KUKA KRL program: f1_Kuka_APT207T03S07.SRC

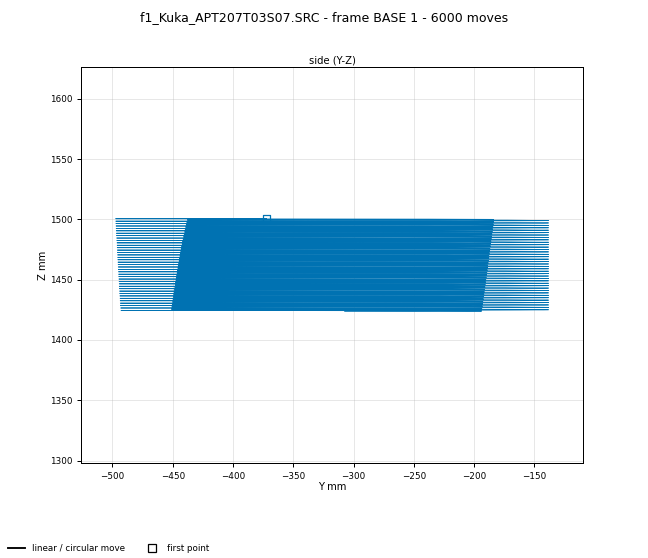
[picture p0: tool path of f1_Kuka_APT207T03S07.SRC in frame BASE 1, 6000 of 6001 moves have a stored position in this frame; points joined in program order, loops and branches not executed]
&ACCESS RVP
&REL 2
&PARAM TEMPLATE = C:\KRC\Roboter\Template\vorgabe
&PARAM EDITMASK = *
DEF f1_Kuka_APT207T03S07()


;FOLD INI;%{PE}%V3.2.0,%MKUKATPBASIS,%CINIT,%VCOMMON,%P
  ;FOLD BAS INI;%{E}%V3.2.0,%MKUKATPBASIS,%CINIT,%VINIT,%P
    GLOBAL INTERRUPT DECL 3 WHEN $STOPMESS==TRUE DO IR_STOPM ( )
    INTERRUPT ON 3
    BAS (#INITMOV,0 )
  ;ENDFOLD (BAS INI)
  ;FOLD USER INI;%{E}%V3.2.0,%MKUKATPUSER,%CINIT,%VINIT,%P
    ;Make your modifications here
  ;ENDFOLD (USER INI)
;ENDFOLD (INI)


;*** Make Null PTP Move
  PTP $pos_act

;*** Auto Load The Correct TOOL Data
  $tool=tool_data[3]

;*** Auto Load The Correct BASE Data
  $base=base_data[1]

  $ADVANCE = 5

;*** Restate Last Velocity
MMPM(30000.0)
SetRPM(6000)
LIN {X 0.159,Y -372.201,Z 1500.629,A 0.000,B 0.000,C 90.000,E1 113.206} C_DIS
LIN {X -0.112,Y -386.220,Z 1500.616,A 0.000,B 0.000,C 90.000,E1 110.918} C_DIS
LIN {X 0.185,Y -401.630,Z 1500.604,A 0.000,B 0.000,C 90.000,E1 108.598} C_DIS
LIN {X 0.113,Y -418.538,Z 1500.591,A 0.000,B 0.000,C 90.000,E1 106.386} C_DIS
LIN {X -0.068,Y -437.063,Z 1500.579,A 0.000,B 0.000,C 90.000,E1 104.245} C_DIS
LIN {X -0.031,Y -456.906,Z 1500.568,A 0.000,B 0.000,C 90.000,E1 102.175} C_DIS
LIN {X 0.162,Y -477.322,Z 1500.557,A 0.000,B 0.000,C 90.000,E1 100.254} C_DIS
LIN {X 0.127,Y -490.260,Z 1500.551,A 0.000,B 0.000,C 90.000,E1 99.151} C_DIS
LIN {X -0.192,Y -492.261,Z 1500.550,A 0.000,B 0.000,C 90.000,E1 98.973} C_DIS
LIN {X 0.126,Y -493.981,Z 1500.548,A 0.000,B 0.000,C 90.000,E1 98.690} C_DIS
LIN {X 0.030,Y -495.267,Z 1500.547,A 0.000,B 0.000,C 90.000,E1 98.454} C_DIS
LIN {X -0.213,Y -496.844,Z 1500.544,A 0.000,B 0.000,C 90.000,E1 97.992} C_DIS
LIN {X 0.043,Y -497.342,Z 1500.542,A 0.000,B 0.000,C 90.000,E1 97.473} C_DIS
LIN {X -0.122,Y -496.847,Z 1500.539,A 0.000,B 0.000,C 90.000,E1 97.004} C_DIS
LIN {X 0.144,Y -495.281,Z 1500.536,A 0.000,B 0.000,C 90.000,E1 96.486} C_DIS
LIN {X 0.002,Y -494.010,Z 1500.535,A 0.000,B 0.000,C 90.000,E1 96.258} C_DIS
LIN {X 0.215,Y -484.168,Z 1500.527,A 0.000,B 0.000,C 90.000,E1 94.759} C_DIS
LIN {X 0.034,Y -473.583,Z 1500.517,A 0.000,B 0.000,C 90.000,E1 93.037} C_DIS
LIN {X 0.219,Y -467.179,Z 1500.511,A 0.000,B 0.000,C 90.000,E1 92.007} C_DIS
LIN {X -0.087,Y -457.018,Z 1500.503,A 0.000,B 0.000,C 90.000,E1 90.516} C_DIS
LIN {X -0.114,Y -446.557,Z 1500.494,A 0.000,B 0.000,C 90.000,E1 88.969} C_DIS
LIN {X 0.127,Y -435.874,Z 1500.485,A 0.000,B 0.000,C 90.000,E1 87.364} C_DIS
LIN {X 0.018,Y -421.489,Z 1500.474,A 0.000,B 0.000,C 90.000,E1 85.241} C_DIS
LIN {X -0.123,Y -410.754,Z 1500.464,A 0.000,B 0.000,C 90.000,E1 83.628} C_DIS
LIN {X 0.119,Y -396.318,Z 1500.452,A 0.000,B 0.000,C 90.000,E1 81.376} C_DIS
LIN {X -0.155,Y -377.030,Z 1500.435,A 0.000,B 0.000,C 90.000,E1 78.285} C_DIS
LIN {X -0.065,Y -363.896,Z 1500.422,A 0.000,B 0.000,C 90.000,E1 75.936} C_DIS
LIN {X -0.051,Y -352.647,Z 1500.410,A 0.000,B 0.000,C 90.000,E1 73.850} C_DIS
LIN {X 0.045,Y -341.368,Z 1500.398,A 0.000,B 0.000,C 90.000,E1 71.710} C_DIS
LIN {X -0.125,Y -328.685,Z 1500.385,A 0.000,B 0.000,C 90.000,E1 69.263} C_DIS
LIN {X 0.116,Y -313.654,Z 1500.367,A 0.000,B 0.000,C 90.000,E1 66.049} C_DIS
LIN {X 0.098,Y -300.896,Z 1500.351,A 0.000,B 0.000,C 90.000,E1 63.127} C_DIS
LIN {X 0.137,Y -288.807,Z 1500.334,A 0.000,B 0.000,C 90.000,E1 60.127} C_DIS
LIN {X -0.069,Y -278.507,Z 1500.319,A 0.000,B 0.000,C 90.000,E1 57.454} C_DIS
LIN {X -0.074,Y -268.552,Z 1500.304,A 0.000,B 0.000,C 90.000,E1 54.689} C_DIS
LIN {X 0.138,Y -258.980,Z 1500.288,A 0.000,B 0.000,C 90.000,E1 51.823} C_DIS
LIN {X 0.047,Y -248.766,Z 1500.270,A 0.000,B 0.000,C 90.000,E1 48.609} C_DIS
LIN {X -0.011,Y -238.232,Z 1500.250,A 0.000,B 0.000,C 90.000,E1 44.960} C_DIS
LIN {X -0.114,Y -230.557,Z 1500.233,A 0.000,B 0.000,C 90.000,E1 42.000} C_DIS
LIN {X -0.005,Y -222.002,Z 1500.212,A 0.000,B 0.000,C 90.000,E1 38.177} C_DIS
LIN {X -0.052,Y -214.472,Z 1500.191,A 0.000,B 0.000,C 90.000,E1 34.326} C_DIS
LIN {X 0.012,Y -207.800,Z 1500.169,A 0.000,B 0.000,C 90.000,E1 30.384} C_DIS
LIN {X -0.013,Y -202.023,Z 1500.147,A 0.000,B 0.000,C 90.000,E1 26.411} C_DIS
LIN {X -0.024,Y -197.120,Z 1500.124,A 0.000,B 0.000,C 90.000,E1 22.386} C_DIS
LIN {X 0.001,Y -192.945,Z 1500.102,A 0.000,B 0.000,C 90.000,E1 18.308} C_DIS
LIN {X 0.065,Y -188.915,Z 1500.074,A 0.000,B 0.000,C 90.000,E1 13.355} C_DIS
LIN {X -0.062,Y -185.704,Z 1500.042,A 0.000,B 0.000,C 90.000,E1 7.587} C_DIS
LIN {X 0.089,Y -183.811,Z 1500.005,A 0.000,B 0.000,C 90.000,E1 0.859} C_DIS
LIN {X -0.056,Y -183.944,Z 1499.965,A 0.000,B 0.000,C 90.000,E1 353.685} C_DIS
LIN {X -0.092,Y -186.302,Z 1499.923,A 0.000,B 0.000,C 90.000,E1 346.172} C_DIS
LIN {X 0.027,Y -189.401,Z 1499.895,A 0.000,B 0.000,C 90.000,E1 341.148} C_DIS
LIN {X -0.076,Y -193.715,Z 1499.868,A 0.000,B 0.000,C 90.000,E1 336.230} C_DIS
LIN {X 0.063,Y -198.267,Z 1499.845,A 0.000,B 0.000,C 90.000,E1 332.103} C_DIS
LIN {X 0.013,Y -203.831,Z 1499.823,A 0.000,B 0.000,C 90.000,E1 328.074} C_DIS
LIN {X -0.061,Y -209.063,Z 1499.805,A 0.000,B 0.000,C 90.000,E1 324.895} C_DIS
LIN {X 0.071,Y -215.145,Z 1499.787,A 0.000,B 0.000,C 90.000,E1 321.698} C_DIS
LIN {X -0.048,Y -222.035,Z 1499.770,A 0.000,B 0.000,C 90.000,E1 318.609} C_DIS
LIN {X -0.009,Y -229.890,Z 1499.753,A 0.000,B 0.000,C 90.000,E1 315.526} C_DIS
LIN {X -0.087,Y -238.715,Z 1499.736,A 0.000,B 0.000,C 90.000,E1 312.528} C_DIS
LIN {X -0.073,Y -249.962,Z 1499.718,A 0.000,B 0.000,C 90.000,E1 309.197} C_DIS
LIN {X 0.003,Y -257.116,Z 1499.708,A 0.000,B 0.000,C 90.000,E1 307.363} C_DIS
LIN {X -0.111,Y -265.197,Z 1499.698,A 0.000,B 0.000,C 90.000,E1 305.598} C_DIS
LIN {X 0.122,Y -274.179,Z 1499.688,A 0.000,B 0.000,C 90.000,E1 303.785} C_DIS
LIN {X -0.024,Y -284.237,Z 1499.678,A 0.000,B 0.000,C 90.000,E1 302.084} C_DIS
LIN {X -0.031,Y -297.487,Z 1499.667,A 0.000,B 0.000,C 90.000,E1 300.050} C_DIS
LIN {X 0.119,Y -307.294,Z 1499.660,A 0.000,B 0.000,C 90.000,E1 298.693} C_DIS
LIN {X 0.060,Y -328.798,Z 1499.646,A 0.000,B 0.000,C 90.000,E1 296.181} C_DIS
LIN {X -0.035,Y -347.607,Z 1499.634,A 0.000,B 0.000,C 90.000,E1 294.207} C_DIS
LIN {X -0.091,Y -363.609,Z 1499.625,A 0.000,B 0.000,C 90.000,E1 292.589} C_DIS
LIN {X -0.201,Y -376.886,Z 1499.618,A 0.000,B 0.000,C 90.000,E1 291.227} C_DIS
LIN {X 0.089,Y -387.250,Z 1499.612,A 0.000,B 0.000,C 90.000,E1 290.066} C_DIS
LIN {X -0.075,Y -397.401,Z 1499.605,A 0.000,B 0.000,C 90.000,E1 288.960} C_DIS
LIN {X -0.160,Y -404.580,Z 1499.601,A 0.000,B 0.000,C 90.000,E1 288.127} C_DIS
LIN {X -0.053,Y -411.214,Z 1499.596,A 0.000,B 0.000,C 90.000,E1 287.275} C_DIS
LIN {X -0.123,Y -415.343,Z 1499.593,A 0.000,B 0.000,C 90.000,E1 286.732} C_DIS
LIN {X -0.046,Y -420.853,Z 1499.588,A 0.000,B 0.000,C 90.000,E1 285.898} C_DIS
LIN {X 0.090,Y -425.661,Z 1499.584,A 0.000,B 0.000,C 90.000,E1 285.064} C_DIS
LIN {X 0.160,Y -429.752,Z 1499.579,A 0.000,B 0.000,C 90.000,E1 284.245} C_DIS
LIN {X 0.094,Y -432.073,Z 1499.576,A 0.000,B 0.000,C 90.000,E1 283.716} C_DIS
LIN {X 0.142,Y -434.062,Z 1499.573,A 0.000,B 0.000,C 90.000,E1 283.175} C_DIS
LIN {X 0.096,Y -435.668,Z 1499.570,A 0.000,B 0.000,C 90.000,E1 282.647} C_DIS
LIN {X 0.060,Y -436.871,Z 1499.567,A 0.000,B 0.000,C 90.000,E1 282.119} C_DIS
LIN {X 0.033,Y -437.649,Z 1499.564,A 0.000,B 0.000,C 90.000,E1 281.591} C_DIS
LIN {X -0.073,Y -437.888,Z 1499.562,A 0.000,B 0.000,C 90.000,E1 281.074} C_DIS
LIN {X -0.087,Y -437.554,Z 1499.558,A 0.000,B 0.000,C 90.000,E1 280.546} C_DIS
LIN {X -0.102,Y -436.689,Z 1499.556,A 0.000,B 0.000,C 90.000,E1 280.018} C_DIS
LIN {X -0.195,Y -435.243,Z 1499.553,A 0.000,B 0.000,C 90.000,E1 279.500} C_DIS
LIN {X 0.209,Y -433.095,Z 1499.550,A 0.000,B 0.000,C 90.000,E1 278.916} C_DIS
LIN {X 0.107,Y -430.136,Z 1499.547,A 0.000,B 0.000,C 90.000,E1 278.398} C_DIS
LIN {X -0.135,Y -428.364,Z 1499.545,A 0.000,B 0.000,C 90.000,E1 278.163} C_DIS
LIN {X 0.159,Y -424.043,Z 1499.542,A 0.000,B 0.000,C 90.000,E1 277.587} C_DIS
LIN {X 0.039,Y -418.760,Z 1499.539,A 0.000,B 0.000,C 90.000,E1 277.068} C_DIS
LIN {X 0.166,Y -412.771,Z 1499.536,A 0.000,B 0.000,C 90.000,E1 276.549} C_DIS
LIN {X -0.111,Y -406.602,Z 1499.534,A 0.000,B 0.000,C 90.000,E1 276.144} C_DIS
LIN {X -0.033,Y -400.296,Z 1499.532,A 0.000,B 0.000,C 90.000,E1 275.739} C_DIS
LIN {X -0.053,Y -393.791,Z 1499.530,A 0.000,B 0.000,C 90.000,E1 275.391} C_DIS
LIN {X -0.100,Y -383.911,Z 1499.527,A 0.000,B 0.000,C 90.000,E1 274.935} C_DIS
LIN {X 0.139,Y -371.250,Z 1499.524,A 0.000,B 0.000,C 90.000,E1 274.359} C_DIS
LIN {X -0.104,Y -358.480,Z 1499.522,A 0.000,B 0.000,C 90.000,E1 273.898} C_DIS
LIN {X -0.130,Y -345.729,Z 1499.519,A 0.000,B 0.000,C 90.000,E1 273.440} C_DIS
LIN {X 0.055,Y -335.630,Z 1499.517,A 0.000,B 0.000,C 90.000,E1 273.094} C_DIS
LIN {X -0.002,Y -322.393,Z 1499.515,A 0.000,B 0.000,C 90.000,E1 272.751} C_DIS
LIN {X -0.068,Y -310.933,Z 1499.514,A 0.000,B 0.000,C 90.000,E1 272.522} C_DIS
LIN {X -0.149,Y -298.734,Z 1499.513,A 0.000,B 0.000,C 90.000,E1 272.350} C_DIS
LIN {X -0.082,Y -287.211,Z 1499.512,A 0.000,B 0.000,C 90.000,E1 272.236} C_DIS
LIN {X 0.016,Y -278.348,Z 1499.512,A 0.000,B 0.000,C 90.000,E1 272.178} C_DIS
LIN {X -0.010,Y -181.234,Z 1499.512,A 0.000,B 0.000,C 90.000,E1 272.178} C_DIS
LIN {X -0.074,Y -181.578,Z 1499.501,A 0.000,B 0.000,C 90.000,E1 270.172} C_DIS
LIN {X -0.085,Y -180.881,Z 1499.473,A 0.000,B 0.000,C 90.000,E1 265.122} C_DIS
LIN {X -0.025,Y -179.000,Z 1499.445,A 0.000,B 0.000,C 90.000,E1 260.038} C_DIS
LIN {X 0.070,Y -178.595,Z 1499.440,A 0.000,B 0.000,C 90.000,E1 259.162} C_DIS
LIN {X -0.037,Y -175.648,Z 1499.412,A 0.000,B 0.000,C 90.000,E1 254.102} C_DIS
LIN {X -0.031,Y -172.366,Z 1499.388,A 0.000,B 0.000,C 90.000,E1 249.826} C_DIS
LIN {X -0.017,Y -171.156,Z 1499.378,A 0.000,B 0.000,C 90.000,E1 248.103} C_DIS
LIN {X 0.028,Y -167.457,Z 1499.354,A 0.000,B 0.000,C 90.000,E1 243.768} C_DIS
LIN {X -0.039,Y -166.853,Z 1499.349,A 0.000,B 0.000,C 90.000,E1 242.922} C_DIS
LIN {X 0.025,Y -162.838,Z 1499.325,A 0.000,B 0.000,C 90.000,E1 238.535} C_DIS
LIN {X 0.000,Y -161.522,Z 1499.315,A 0.000,B 0.000,C 90.000,E1 236.786} C_DIS
LIN {X 0.041,Y -157.521,Z 1499.291,A 0.000,B 0.000,C 90.000,E1 232.351} C_DIS
LIN {X -0.026,Y -155.545,Z 1499.276,A 0.000,B 0.000,C 90.000,E1 229.703} C_DIS
LIN {X 0.016,Y -151.838,Z 1499.251,A 0.000,B 0.000,C 90.000,E1 225.202} C_DIS
LIN {X -0.077,Y -150.056,Z 1499.236,A 0.000,B 0.000,C 90.000,E1 222.528} C_DIS
LIN {X 0.048,Y -146.868,Z 1499.211,A 0.000,B 0.000,C 90.000,E1 217.935} C_DIS
LIN {X -0.053,Y -145.452,Z 1499.196,A 0.000,B 0.000,C 90.000,E1 215.231} C_DIS
LIN {X 0.061,Y -142.869,Z 1499.170,A 0.000,B 0.000,C 90.000,E1 210.590} C_DIS
LIN {X -0.013,Y -141.487,Z 1499.150,A 0.000,B 0.000,C 90.000,E1 206.924} C_DIS
LIN {X -0.028,Y -139.383,Z 1499.113,A 0.000,B 0.000,C 90.000,E1 200.429} C_DIS
LIN {X -0.040,Y -138.839,Z 1499.098,A 0.000,B 0.000,C 90.000,E1 197.638} C_DIS
LIN {X 0.021,Y -138.354,Z 1499.056,A 0.000,B 0.000,C 90.000,E1 190.141} C_DIS
LIN {X 0.016,Y -139.522,Z 1499.005,A 0.000,B 0.000,C 90.000,E1 180.802} C_DIS
LIN {X -0.043,Y -141.185,Z 1498.974,A 0.000,B 0.000,C 90.000,E1 175.241} C_DIS
LIN {X 0.069,Y -142.563,Z 1498.958,A 0.000,B 0.000,C 90.000,E1 172.413} C_DIS
LIN {X 0.024,Y -144.847,Z 1498.932,A 0.000,B 0.000,C 90.000,E1 167.813} C_DIS
LIN {X -0.020,Y -147.472,Z 1498.912,A 0.000,B 0.000,C 90.000,E1 164.157} C_DIS
LIN {X 0.006,Y -150.056,Z 1498.892,A 0.000,B 0.000,C 90.000,E1 160.496} C_DIS
LIN {X 0.011,Y -153.401,Z 1498.871,A 0.000,B 0.000,C 90.000,E1 156.869} C_DIS
LIN {X 0.057,Y -155.931,Z 1498.857,A 0.000,B 0.000,C 90.000,E1 154.152} C_DIS
LIN {X 0.031,Y -159.799,Z 1498.837,A 0.000,B 0.000,C 90.000,E1 150.589} C_DIS
LIN {X 0.016,Y -162.040,Z 1498.827,A 0.000,B 0.000,C 90.000,E1 148.820} C_DIS
LIN {X -0.009,Y -166.235,Z 1498.807,A 0.000,B 0.000,C 90.000,E1 145.308} C_DIS
LIN {X -0.007,Y -171.251,Z 1498.788,A 0.000,B 0.000,C 90.000,E1 141.823} C_DIS
LIN {X -0.086,Y -176.141,Z 1498.769,A 0.000,B 0.000,C 90.000,E1 138.405} C_DIS
LIN {X 0.031,Y -180.408,Z 1498.755,A 0.000,B 0.000,C 90.000,E1 135.810} C_DIS
LIN {X 0.006,Y -185.815,Z 1498.736,A 0.000,B 0.000,C 90.000,E1 132.447} C_DIS
LIN {X 0.061,Y -190.434,Z 1498.722,A 0.000,B 0.000,C 90.000,E1 129.930} C_DIS
LIN {X 0.113,Y -197.759,Z 1498.699,A 0.000,B 0.000,C 90.000,E1 125.804} C_DIS
LIN {X -0.115,Y -201.427,Z 1498.689,A 0.000,B 0.000,C 90.000,E1 123.992} C_DIS
LIN {X -0.117,Y -201.783,Z 1498.688,A 0.000,B 0.000,C 90.000,E1 123.785} C_DIS
LIN {X 0.201,Y -315.841,Z 1498.688,A 0.000,B 0.000,C 90.000,E1 123.706} C_DIS
LIN {X 0.042,Y -317.337,Z 1498.687,A 0.000,B 0.000,C 90.000,E1 123.706} C_DIS
LIN {X -0.100,Y -323.116,Z 1498.686,A 0.000,B 0.000,C 90.000,E1 123.420} C_DIS
LIN {X -0.079,Y -326.279,Z 1498.684,A 0.000,B 0.000,C 90.000,E1 123.086} C_DIS
LIN {X 0.187,Y -328.261,Z 1498.682,A 0.000,B 0.000,C 90.000,E1 122.752} C_DIS
LIN {X 0.003,Y -329.813,Z 1498.681,A 0.000,B 0.000,C 90.000,E1 122.498} C_DIS
LIN {X -0.055,Y -332.315,Z 1498.677,A 0.000,B 0.000,C 90.000,E1 121.878} C_DIS
LIN {X -0.045,Y -343.419,Z 1498.661,A 0.000,B 0.000,C 90.000,E1 119.077} C_DIS
LIN {X 0.089,Y -355.915,Z 1498.646,A 0.000,B 0.000,C 90.000,E1 116.309} C_DIS
LIN {X -0.046,Y -369.903,Z 1498.631,A 0.000,B 0.000,C 90.000,E1 113.643} C_DIS
LIN {X 0.117,Y -383.694,Z 1498.618,A 0.000,B 0.000,C 90.000,E1 111.280} C_DIS
LIN {X -0.151,Y -398.857,Z 1498.606,A 0.000,B 0.000,C 90.000,E1 109.033} C_DIS
LIN {X -0.177,Y -415.499,Z 1498.593,A 0.000,B 0.000,C 90.000,E1 106.804} C_DIS
LIN {X 0.086,Y -433.737,Z 1498.581,A 0.000,B 0.000,C 90.000,E1 104.592} C_DIS
LIN {X -0.166,Y -453.418,Z 1498.570,A 0.000,B 0.000,C 90.000,E1 102.535} C_DIS
LIN {X -0.113,Y -473.742,Z 1498.559,A 0.000,B 0.000,C 90.000,E1 100.602} C_DIS
LIN {X -0.154,Y -489.320,Z 1498.551,A 0.000,B 0.000,C 90.000,E1 99.265} C_DIS
LIN {X 0.005,Y -491.539,Z 1498.550,A 0.000,B 0.000,C 90.000,E1 99.029} C_DIS
LIN {X -0.110,Y -493.374,Z 1498.549,A 0.000,B 0.000,C 90.000,E1 98.803} C_DIS
LIN {X -0.149,Y -494.756,Z 1498.547,A 0.000,B 0.000,C 90.000,E1 98.568} C_DIS
LIN {X 0.093,Y -496.549,Z 1498.545,A 0.000,B 0.000,C 90.000,E1 98.049} C_DIS
LIN {X -0.146,Y -497.227,Z 1498.542,A 0.000,B 0.000,C 90.000,E1 97.587} C_DIS
LIN {X 0.118,Y -496.908,Z 1498.539,A 0.000,B 0.000,C 90.000,E1 97.068} C_DIS
LIN {X -0.106,Y -495.545,Z 1498.537,A 0.000,B 0.000,C 90.000,E1 96.606} C_DIS
LIN {X -0.191,Y -494.403,Z 1498.535,A 0.000,B 0.000,C 90.000,E1 96.372} C_DIS
LIN {X 0.064,Y -491.104,Z 1498.533,A 0.000,B 0.000,C 90.000,E1 95.853} C_DIS
LIN {X -0.128,Y -483.063,Z 1498.526,A 0.000,B 0.000,C 90.000,E1 94.645} C_DIS
LIN {X 0.147,Y -472.480,Z 1498.516,A 0.000,B 0.000,C 90.000,E1 92.865} C_DIS
LIN {X 0.133,Y -464.318,Z 1498.509,A 0.000,B 0.000,C 90.000,E1 91.604} C_DIS
LIN {X 0.225,Y -454.111,Z 1498.500,A 0.000,B 0.000,C 90.000,E1 90.057} C_DIS
LIN {X 0.139,Y -443.573,Z 1498.492,A 0.000,B 0.000,C 90.000,E1 88.511} C_DIS
LIN {X -0.115,Y -432.845,Z 1498.483,A 0.000,B 0.000,C 90.000,E1 86.963} C_DIS
LIN {X 0.162,Y -418.583,Z 1498.471,A 0.000,B 0.000,C 90.000,E1 84.780} C_DIS
LIN {X 0.079,Y -406.016,Z 1498.460,A 0.000,B 0.000,C 90.000,E1 82.875} C_DIS
LIN {X -0.185,Y -391.653,Z 1498.448,A 0.000,B 0.000,C 90.000,E1 80.679} C_DIS
LIN {X -0.141,Y -372.690,Z 1498.431,A 0.000,B 0.000,C 90.000,E1 77.521} C_DIS
LIN {X -0.156,Y -359.715,Z 1498.417,A 0.000,B 0.000,C 90.000,E1 75.172} C_DIS
LIN {X 0.095,Y -348.455,Z 1498.406,A 0.000,B 0.000,C 90.000,E1 73.032} C_DIS
LIN {X -0.017,Y -337.208,Z 1498.394,A 0.000,B 0.000,C 90.000,E1 70.913} C_DIS
LIN {X -0.016,Y -323.150,Z 1498.378,A 0.000,B 0.000,C 90.000,E1 68.103} C_DIS
LIN {X -0.117,Y -308.449,Z 1498.361,A 0.000,B 0.000,C 90.000,E1 64.921} C_DIS
LIN {X -0.138,Y -295.967,Z 1498.344,A 0.000,B 0.000,C 90.000,E1 61.975} C_DIS
LIN {X -0.091,Y -284.131,Z 1498.327,A 0.000,B 0.000,C 90.000,E1 58.948} C_DIS
LIN {X -0.110,Y -274.017,Z 1498.312,A 0.000,B 0.000,C 90.000,E1 56.215} C_DIS
LIN {X -0.002,Y -263.059,Z 1498.295,A 0.000,B 0.000,C 90.000,E1 53.050} C_DIS
LIN {X 0.056,Y -252.637,Z 1498.277,A 0.000,B 0.000,C 90.000,E1 49.828} C_DIS
LIN {X -0.047,Y -242.911,Z 1498.259,A 0.000,B 0.000,C 90.000,E1 46.581} C_DIS
LIN {X -0.041,Y -234.847,Z 1498.242,A 0.000,B 0.000,C 90.000,E1 43.623} C_DIS
LIN {X -0.050,Y -227.584,Z 1498.226,A 0.000,B 0.000,C 90.000,E1 40.620} C_DIS
LIN {X -0.045,Y -220.937,Z 1498.209,A 0.000,B 0.000,C 90.000,E1 37.569} C_DIS
LIN {X -0.078,Y -213.560,Z 1498.187,A 0.000,B 0.000,C 90.000,E1 33.706} C_DIS
LIN {X 0.030,Y -207.020,Z 1498.165,A 0.000,B 0.000,C 90.000,E1 29.745} C_DIS
LIN {X -0.014,Y -201.412,Z 1498.143,A 0.000,B 0.000,C 90.000,E1 25.771} C_DIS
LIN {X 0.060,Y -196.654,Z 1498.121,A 0.000,B 0.000,C 90.000,E1 21.716} C_DIS
LIN {X 0.070,Y -192.592,Z 1498.098,A 0.000,B 0.000,C 90.000,E1 17.638} C_DIS
LIN {X 0.022,Y -188.726,Z 1498.071,A 0.000,B 0.000,C 90.000,E1 12.715} C_DIS
LIN {X 0.073,Y -185.715,Z 1498.038,A 0.000,B 0.000,C 90.000,E1 6.891} C_DIS
LIN {X -0.033,Y -183.948,Z 1497.997,A 0.000,B 0.000,C 90.000,E1 359.542} C_DIS
LIN {X 0.052,Y -184.347,Z 1497.960,A 0.000,B 0.000,C 90.000,E1 352.818} C_DIS
LIN {X -0.065,Y -186.532,Z 1497.923,A 0.000,B 0.000,C 90.000,E1 346.172} C_DIS
LIN {X 0.062,Y -189.608,Z 1497.895,A 0.000,B 0.000,C 90.000,E1 341.148} C_DIS
LIN {X -0.033,Y -193.892,Z 1497.868,A 0.000,B 0.000,C 90.000,E1 336.230} C_DIS
LIN {X -0.064,Y -198.427,Z 1497.845,A 0.000,B 0.000,C 90.000,E1 332.153} C_DIS
LIN {X 0.100,Y -202.767,Z 1497.827,A 0.000,B 0.000,C 90.000,E1 328.869} C_DIS
LIN {X 0.061,Y -207.818,Z 1497.809,A 0.000,B 0.000,C 90.000,E1 325.674} C_DIS
LIN {X -0.135,Y -213.673,Z 1497.792,A 0.000,B 0.000,C 90.000,E1 322.557} C_DIS
LIN {X 0.041,Y -220.355,Z 1497.774,A 0.000,B 0.000,C 90.000,E1 319.380} C_DIS
LIN {X 0.036,Y -227.975,Z 1497.757,A 0.000,B 0.000,C 90.000,E1 316.296} C_DIS
LIN {X 0.032,Y -237.714,Z 1497.738,A 0.000,B 0.000,C 90.000,E1 312.894} C_DIS
LIN {X 0.014,Y -248.788,Z 1497.720,A 0.000,B 0.000,C 90.000,E1 309.564} C_DIS
LIN {X 0.101,Y -257.255,Z 1497.708,A 0.000,B 0.000,C 90.000,E1 307.363} C_DIS
LIN {X -0.008,Y -265.305,Z 1497.698,A 0.000,B 0.000,C 90.000,E1 305.598} C_DIS
LIN {X 0.002,Y -274.232,Z 1497.688,A 0.000,B 0.000,C 90.000,E1 303.833} C_DIS
LIN {X 0.045,Y -286.338,Z 1497.676,A 0.000,B 0.000,C 90.000,E1 301.750} C_DIS
LIN {X -0.062,Y -297.390,Z 1497.667,A 0.000,B 0.000,C 90.000,E1 300.079} C_DIS
LIN {X 0.032,Y -307.080,Z 1497.660,A 0.000,B 0.000,C 90.000,E1 298.743} C_DIS
LIN {X -0.047,Y -328.124,Z 1497.646,A 0.000,B 0.000,C 90.000,E1 296.283} C_DIS
LIN {X -0.131,Y -347.427,Z 1497.635,A 0.000,B 0.000,C 90.000,E1 294.259} C_DIS
LIN {X 0.093,Y -363.526,Z 1497.626,A 0.000,B 0.000,C 90.000,E1 292.589} C_DIS
LIN {X 0.131,Y -376.594,Z 1497.618,A 0.000,B 0.000,C 90.000,E1 291.227} C_DIS
LIN {X 0.115,Y -386.924,Z 1497.612,A 0.000,B 0.000,C 90.000,E1 290.120} C_DIS
LIN {X -0.150,Y -397.085,Z 1497.606,A 0.000,B 0.000,C 90.000,E1 289.033} C_DIS
LIN {X -0.111,Y -404.328,Z 1497.601,A 0.000,B 0.000,C 90.000,E1 288.181} C_DIS
LIN {X -0.006,Y -411.014,Z 1497.596,A 0.000,B 0.000,C 90.000,E1 287.330} C_DIS
LIN {X 0.032,Y -417.083,Z 1497.592,A 0.000,B 0.000,C 90.000,E1 286.496} C_DIS
LIN {X 0.135,Y -422.487,Z 1497.587,A 0.000,B 0.000,C 90.000,E1 285.662} C_DIS
LIN {X -0.129,Y -427.145,Z 1497.583,A 0.000,B 0.000,C 90.000,E1 284.883} C_DIS
LIN {X -0.044,Y -431.058,Z 1497.578,A 0.000,B 0.000,C 90.000,E1 284.064} C_DIS
LIN {X 0.081,Y -434.215,Z 1497.574,A 0.000,B 0.000,C 90.000,E1 283.244} C_DIS
LIN {X 0.037,Y -435.908,Z 1497.571,A 0.000,B 0.000,C 90.000,E1 282.715} C_DIS
LIN {X 0.006,Y -437.212,Z 1497.568,A 0.000,B 0.000,C 90.000,E1 282.187} C_DIS
LIN {X -0.017,Y -438.061,Z 1497.565,A 0.000,B 0.000,C 90.000,E1 281.658} C_DIS
LIN {X -0.032,Y -438.379,Z 1497.562,A 0.000,B 0.000,C 90.000,E1 281.130} C_DIS
LIN {X -0.046,Y -438.162,Z 1497.559,A 0.000,B 0.000,C 90.000,E1 280.602} C_DIS
LIN {X -0.059,Y -437.398,Z 1497.556,A 0.000,B 0.000,C 90.000,E1 280.074} C_DIS
LIN {X -0.149,Y -436.003,Z 1497.553,A 0.000,B 0.000,C 90.000,E1 279.557} C_DIS
LIN {X -0.169,Y -433.970,Z 1497.550,A 0.000,B 0.000,C 90.000,E1 279.029} C_DIS
LIN {X -0.038,Y -432.698,Z 1497.549,A 0.000,B 0.000,C 90.000,E1 278.746} C_DIS
LIN {X -0.080,Y -429.413,Z 1497.546,A 0.000,B 0.000,C 90.000,E1 278.219} C_DIS
LIN {X -0.202,Y -425.288,Z 1497.543,A 0.000,B 0.000,C 90.000,E1 277.701} C_DIS
LIN {X 0.076,Y -420.087,Z 1497.540,A 0.000,B 0.000,C 90.000,E1 277.125} C_DIS
LIN {X 0.152,Y -414.169,Z 1497.537,A 0.000,B 0.000,C 90.000,E1 276.606} C_DIS
LIN {X -0.176,Y -408.000,Z 1497.534,A 0.000,B 0.000,C 90.000,E1 276.201} C_DIS
LIN {X -0.153,Y -401.649,Z 1497.532,A 0.000,B 0.000,C 90.000,E1 275.796} C_DIS
LIN {X 0.181,Y -395.109,Z 1497.530,A 0.000,B 0.000,C 90.000,E1 275.391} C_DIS
LIN {X 0.127,Y -385.320,Z 1497.527,A 0.000,B 0.000,C 90.000,E1 274.935} C_DIS
LIN {X -0.039,Y -372.681,Z 1497.525,A 0.000,B 0.000,C 90.000,E1 274.416} C_DIS
LIN {X 0.025,Y -359.675,Z 1497.522,A 0.000,B 0.000,C 90.000,E1 273.898} C_DIS
LIN {X -0.027,Y -346.895,Z 1497.519,A 0.000,B 0.000,C 90.000,E1 273.440} C_DIS
LIN {X 0.136,Y -336.792,Z 1497.517,A 0.000,B 0.000,C 90.000,E1 273.094} C_DIS
LIN {X 0.053,Y -323.310,Z 1497.515,A 0.000,B 0.000,C 90.000,E1 272.751} C_DIS
LIN {X -0.023,Y -312.085,Z 1497.514,A 0.000,B 0.000,C 90.000,E1 272.522} C_DIS
LIN {X -0.117,Y -299.722,Z 1497.513,A 0.000,B 0.000,C 90.000,E1 272.350} C_DIS
LIN {X -0.051,Y -288.421,Z 1497.512,A 0.000,B 0.000,C 90.000,E1 272.236} C_DIS
LIN {X 0.043,Y -279.019,Z 1497.512,A 0.000,B 0.000,C 90.000,E1 272.178} C_DIS
LIN {X 0.008,Y -181.233,Z 1497.512,A 0.000,B 0.000,C 90.000,E1 272.178} C_DIS
LIN {X -0.057,Y -181.578,Z 1497.501,A 0.000,B 0.000,C 90.000,E1 270.172} C_DIS
LIN {X -0.067,Y -180.882,Z 1497.473,A 0.000,B 0.000,C 90.000,E1 265.122} C_DIS
LIN {X -0.007,Y -179.001,Z 1497.445,A 0.000,B 0.000,C 90.000,E1 260.038} C_DIS
LIN {X 0.087,Y -178.599,Z 1497.440,A 0.000,B 0.000,C 90.000,E1 259.162} C_DIS
LIN {X -0.021,Y -175.651,Z 1497.412,A 0.000,B 0.000,C 90.000,E1 254.102} C_DIS
LIN {X -0.014,Y -172.370,Z 1497.388,A 0.000,B 0.000,C 90.000,E1 249.826} C_DIS
LIN {X 0.000,Y -171.163,Z 1497.378,A 0.000,B 0.000,C 90.000,E1 248.103} C_DIS
LIN {X 0.043,Y -167.461,Z 1497.354,A 0.000,B 0.000,C 90.000,E1 243.768} C_DIS
LIN {X -0.023,Y -166.856,Z 1497.349,A 0.000,B 0.000,C 90.000,E1 242.922} C_DIS
LIN {X 0.042,Y -162.842,Z 1497.325,A 0.000,B 0.000,C 90.000,E1 238.535} C_DIS
LIN {X 0.016,Y -161.526,Z 1497.316,A 0.000,B 0.000,C 90.000,E1 236.786} C_DIS
LIN {X 0.057,Y -157.526,Z 1497.291,A 0.000,B 0.000,C 90.000,E1 232.351} C_DIS
LIN {X -0.011,Y -155.550,Z 1497.276,A 0.000,B 0.000,C 90.000,E1 229.703} C_DIS
LIN {X -0.076,Y -151.842,Z 1497.251,A 0.000,B 0.000,C 90.000,E1 225.243} C_DIS
LIN {X -0.062,Y -150.060,Z 1497.236,A 0.000,B 0.000,C 90.000,E1 222.528} C_DIS
LIN {X -0.027,Y -146.871,Z 1497.211,A 0.000,B 0.000,C 90.000,E1 217.971} C_DIS
LIN {X -0.038,Y -145.457,Z 1497.196,A 0.000,B 0.000,C 90.000,E1 215.231} C_DIS
LIN {X 0.075,Y -142.872,Z 1497.170,A 0.000,B 0.000,C 90.000,E1 210.590} C_DIS
LIN {X 0.001,Y -141.490,Z 1497.150,A 0.000,B 0.000,C 90.000,E1 206.924} C_DIS
LIN {X -0.014,Y -139.384,Z 1497.113,A 0.000,B 0.000,C 90.000,E1 200.429} C_DIS
LIN {X -0.025,Y -138.840,Z 1497.098,A 0.000,B 0.000,C 90.000,E1 197.638} C_DIS
LIN {X 0.035,Y -138.354,Z 1497.056,A 0.000,B 0.000,C 90.000,E1 190.141} C_DIS
LIN {X 0.031,Y -139.521,Z 1497.005,A 0.000,B 0.000,C 90.000,E1 180.802} C_DIS
LIN {X -0.028,Y -141.183,Z 1496.974,A 0.000,B 0.000,C 90.000,E1 175.241} C_DIS
LIN {X -0.058,Y -142.561,Z 1496.958,A 0.000,B 0.000,C 90.000,E1 172.470} C_DIS
LIN {X 0.009,Y -144.843,Z 1496.932,A 0.000,B 0.000,C 90.000,E1 167.825} C_DIS
LIN {X -0.005,Y -147.467,Z 1496.912,A 0.000,B 0.000,C 90.000,E1 164.157} C_DIS
LIN {X 0.021,Y -150.052,Z 1496.892,A 0.000,B 0.000,C 90.000,E1 160.496} C_DIS
LIN {X 0.027,Y -153.395,Z 1496.872,A 0.000,B 0.000,C 90.000,E1 156.869} C_DIS
LIN {X 0.073,Y -155.925,Z 1496.857,A 0.000,B 0.000,C 90.000,E1 154.152} C_DIS
LIN {X 0.047,Y -159.792,Z 1496.837,A 0.000,B 0.000,C 90.000,E1 150.589} C_DIS
LIN {X 0.033,Y -162.032,Z 1496.827,A 0.000,B 0.000,C 90.000,E1 148.820} C_DIS
LIN {X 0.007,Y -166.228,Z 1496.807,A 0.000,B 0.000,C 90.000,E1 145.308} C_DIS
LIN {X 0.009,Y -171.244,Z 1496.788,A 0.000,B 0.000,C 90.000,E1 141.823} C_DIS
LIN {X -0.068,Y -176.132,Z 1496.769,A 0.000,B 0.000,C 90.000,E1 138.405} C_DIS
LIN {X 0.048,Y -180.399,Z 1496.755,A 0.000,B 0.000,C 90.000,E1 135.810} C_DIS
LIN {X 0.024,Y -185.806,Z 1496.736,A 0.000,B 0.000,C 90.000,E1 132.447} C_DIS
LIN {X 0.079,Y -190.424,Z 1496.722,A 0.000,B 0.000,C 90.000,E1 129.930} C_DIS
LIN {X -0.030,Y -197.749,Z 1496.699,A 0.000,B 0.000,C 90.000,E1 125.851} C_DIS
LIN {X -0.096,Y -201.419,Z 1496.689,A 0.000,B 0.000,C 90.000,E1 123.992} C_DIS
LIN {X 0.018,Y -201.718,Z 1496.688,A 0.000,B 0.000,C 90.000,E1 123.785} C_DIS
LIN {X -0.032,Y -315.212,Z 1496.688,A 0.000,B 0.000,C 90.000,E1 123.785} C_DIS
LIN {X -0.153,Y -316.677,Z 1496.688,A 0.000,B 0.000,C 90.000,E1 123.785} C_DIS
LIN {X 0.022,Y -320.933,Z 1496.687,A 0.000,B 0.000,C 90.000,E1 123.579} C_DIS
LIN {X -0.071,Y -323.288,Z 1496.686,A 0.000,B 0.000,C 90.000,E1 123.420} C_DIS
LIN {X 0.055,Y -327.141,Z 1496.683,A 0.000,B 0.000,C 90.000,E1 122.959} C_DIS
LIN {X -0.062,Y -329.001,Z 1496.682,A 0.000,B 0.000,C 90.000,E1 122.673} C_DIS
LIN {X 0.098,Y -330.456,Z 1496.680,A 0.000,B 0.000,C 90.000,E1 122.339} C_DIS
LIN {X -0.107,Y -343.987,Z 1496.661,A 0.000,B 0.000,C 90.000,E1 118.949} C_DIS
LIN {X 0.043,Y -356.555,Z 1496.646,A 0.000,B 0.000,C 90.000,E1 116.181} C_DIS
LIN {X -0.078,Y -370.621,Z 1496.631,A 0.000,B 0.000,C 90.000,E1 113.515} C_DIS
LIN {X 0.101,Y -384.485,Z 1496.618,A 0.000,B 0.000,C 90.000,E1 111.153} C_DIS
LIN {X -0.152,Y -399.729,Z 1496.605,A 0.000,B 0.000,C 90.000,E1 108.906} C_DIS
LIN {X -0.162,Y -416.457,Z 1496.593,A 0.000,B 0.000,C 90.000,E1 106.677} C_DIS
LIN {X 0.010,Y -434.787,Z 1496.580,A 0.000,B 0.000,C 90.000,E1 104.481} C_DIS
LIN {X -0.082,Y -454.527,Z 1496.569,A 0.000,B 0.000,C 90.000,E1 102.411} C_DIS
LIN {X -0.047,Y -474.881,Z 1496.558,A 0.000,B 0.000,C 90.000,E1 100.489} C_DIS
LIN {X -0.027,Y -490.368,Z 1496.551,A 0.000,B 0.000,C 90.000,E1 99.151} C_DIS
LIN {X 0.141,Y -492.292,Z 1496.550,A 0.000,B 0.000,C 90.000,E1 98.916} C_DIS
LIN {X 0.046,Y -493.953,Z 1496.548,A 0.000,B 0.000,C 90.000,E1 98.681} C_DIS
LIN {X -0.124,Y -495.194,Z 1496.547,A 0.000,B 0.000,C 90.000,E1 98.454} C_DIS
LIN {X 0.124,Y -496.702,Z 1496.544,A 0.000,B 0.000,C 90.000,E1 97.936} C_DIS
LIN {X -0.048,Y -497.140,Z 1496.542,A 0.000,B 0.000,C 90.000,E1 97.466} C_DIS
LIN {X 0.214,Y -496.586,Z 1496.539,A 0.000,B 0.000,C 90.000,E1 96.947} C_DIS
LIN {X -0.013,Y -494.950,Z 1496.536,A 0.000,B 0.000,C 90.000,E1 96.486} C_DIS
LIN {X -0.155,Y -493.636,Z 1496.535,A 0.000,B 0.000,C 90.000,E1 96.258} C_DIS
LIN {X 0.175,Y -485.305,Z 1496.528,A 0.000,B 0.000,C 90.000,E1 94.992} C_DIS
LIN {X -0.130,Y -473.186,Z 1496.517,A 0.000,B 0.000,C 90.000,E1 93.037} C_DIS
LIN {X -0.135,Y -465.111,Z 1496.510,A 0.000,B 0.000,C 90.000,E1 91.776} C_DIS
LIN {X -0.025,Y -454.922,Z 1496.501,A 0.000,B 0.000,C 90.000,E1 90.229} C_DIS
LIN {X -0.090,Y -444.426,Z 1496.493,A 0.000,B 0.000,C 90.000,E1 88.682} C_DIS
LIN {X 0.111,Y -433.757,Z 1496.484,A 0.000,B 0.000,C 90.000,E1 87.078} C_DIS
LIN {X -0.015,Y -419.520,Z 1496.472,A 0.000,B 0.000,C 90.000,E1 84.951} C_DIS
LIN {X -0.114,Y -407.018,Z 1496.461,A 0.000,B 0.000,C 90.000,E1 83.053} C_DIS
LIN {X 0.095,Y -392.668,Z 1496.449,A 0.000,B 0.000,C 90.000,E1 80.792} C_DIS
LIN {X 0.089,Y -371.995,Z 1496.430,A 0.000,B 0.000,C 90.000,E1 77.353} C_DIS
LIN {X 0.132,Y -359.034,Z 1496.417,A 0.000,B 0.000,C 90.000,E1 74.991} C_DIS
LIN {X 0.028,Y -347.775,Z 1496.405,A 0.000,B 0.000,C 90.000,E1 72.906} C_DIS
LIN {X -0.092,Y -336.503,Z 1496.393,A 0.000,B 0.000,C 90.000,E1 70.786} C_DIS
LIN {X -0.102,Y -322.468,Z 1496.378,A 0.000,B 0.000,C 90.000,E1 67.975} C_DIS
LIN {X 0.192,Y -307.804,Z 1496.360,A 0.000,B 0.000,C 90.000,E1 64.717} C_DIS
LIN {X 0.148,Y -295.391,Z 1496.343,A 0.000,B 0.000,C 90.000,E1 61.769} C_DIS
LIN {X -0.069,Y -283.600,Z 1496.327,A 0.000,B 0.000,C 90.000,E1 58.791} C_DIS
LIN {X 0.133,Y -273.525,Z 1496.311,A 0.000,B 0.000,C 90.000,E1 56.008} C_DIS
LIN {X 0.006,Y -262.634,Z 1496.294,A 0.000,B 0.000,C 90.000,E1 52.889} C_DIS
LIN {X 0.083,Y -251.160,Z 1496.274,A 0.000,B 0.000,C 90.000,E1 49.299} C_DIS
LIN {X 0.095,Y -240.554,Z 1496.254,A 0.000,B 0.000,C 90.000,E1 45.648} C_DIS
LIN {X 0.040,Y -232.735,Z 1496.237,A 0.000,B 0.000,C 90.000,E1 42.690} C_DIS
LIN {X 0.038,Y -224.028,Z 1496.216,A 0.000,B 0.000,C 90.000,E1 38.910} C_DIS
LIN {X -0.013,Y -217.763,Z 1496.199,A 0.000,B 0.000,C 90.000,E1 35.851} C_DIS
LIN {X 0.086,Y -210.763,Z 1496.177,A 0.000,B 0.000,C 90.000,E1 31.926} C_DIS
LIN {X 0.073,Y -204.654,Z 1496.156,A 0.000,B 0.000,C 90.000,E1 27.975} C_DIS
LIN {X -0.049,Y -199.445,Z 1496.133,A 0.000,B 0.000,C 90.000,E1 24.003} C_DIS
LIN {X -0.002,Y -195.007,Z 1496.111,A 0.000,B 0.000,C 90.000,E1 19.939} C_DIS
LIN {X 0.061,Y -190.653,Z 1496.083,A 0.000,B 0.000,C 90.000,E1 15.009} C_DIS
LIN {X -0.013,Y -187.456,Z 1496.056,A 0.000,B 0.000,C 90.000,E1 10.074} C_DIS
LIN {X -0.090,Y -184.856,Z 1496.019,A 0.000,B 0.000,C 90.000,E1 3.440} C_DIS
LIN {X 0.083,Y -184.185,Z 1495.979,A 0.000,B 0.000,C 90.000,E1 356.159} C_DIS
LIN {X 0.002,Y -185.178,Z 1495.946,A 0.000,B 0.000,C 90.000,E1 350.330} C_DIS
LIN {X -0.076,Y -187.627,Z 1495.914,A 0.000,B 0.000,C 90.000,E1 344.519} C_DIS
LIN {X 0.021,Y -191.106,Z 1495.886,A 0.000,B 0.000,C 90.000,E1 339.518} C_DIS
LIN {X 0.012,Y -194.892,Z 1495.863,A 0.000,B 0.000,C 90.000,E1 335.409} C_DIS
LIN {X 0.105,Y -199.574,Z 1495.841,A 0.000,B 0.000,C 90.000,E1 331.307} C_DIS
LIN {X -0.075,Y -205.336,Z 1495.818,A 0.000,B 0.000,C 90.000,E1 327.327} C_DIS
LIN {X 0.008,Y -210.786,Z 1495.801,A 0.000,B 0.000,C 90.000,E1 324.116} C_DIS
LIN {X 0.014,Y -217.052,Z 1495.783,A 0.000,B 0.000,C 90.000,E1 320.964} C_DIS
LIN {X -0.062,Y -224.180,Z 1495.766,A 0.000,B 0.000,C 90.000,E1 317.877} C_DIS
LIN {X 0.025,Y -232.324,Z 1495.749,A 0.000,B 0.000,C 90.000,E1 314.798} C_DIS
LIN {X -0.152,Y -241.428,Z 1495.732,A 0.000,B 0.000,C 90.000,E1 311.838} C_DIS
LIN {X 0.112,Y -250.282,Z 1495.718,A 0.000,B 0.000,C 90.000,E1 309.197} C_DIS
LIN {X 0.043,Y -257.408,Z 1495.708,A 0.000,B 0.000,C 90.000,E1 307.397} C_DIS
LIN {X 0.147,Y -267.122,Z 1495.696,A 0.000,B 0.000,C 90.000,E1 305.231} C_DIS
LIN {X -0.043,Y -274.300,Z 1495.688,A 0.000,B 0.000,C 90.000,E1 303.865} C_DIS
LIN {X -0.085,Y -286.329,Z 1495.677,A 0.000,B 0.000,C 90.000,E1 301.799} C_DIS
LIN {X 0.057,Y -297.342,Z 1495.667,A 0.000,B 0.000,C 90.000,E1 300.079} C_DIS
LIN {X 0.133,Y -307.002,Z 1495.660,A 0.000,B 0.000,C 90.000,E1 298.743} C_DIS
LIN {X 0.117,Y -328.428,Z 1495.646,A 0.000,B 0.000,C 90.000,E1 296.232} C_DIS
LIN {X 0.110,Y -347.724,Z 1495.635,A 0.000,B 0.000,C 90.000,E1 294.207} C_DIS
LIN {X -0.202,Y -361.167,Z 1495.627,A 0.000,B 0.000,C 90.000,E1 292.898} C_DIS
LIN {X 0.042,Y -371.738,Z 1495.621,A 0.000,B 0.000,C 90.000,E1 291.770} C_DIS
LIN {X 0.090,Y -382.151,Z 1495.615,A 0.000,B 0.000,C 90.000,E1 290.663} C_DIS
LIN {X -0.143,Y -392.428,Z 1495.609,A 0.000,B 0.000,C 90.000,E1 289.577} C_DIS
LIN {X -0.078,Y -399.936,Z 1495.604,A 0.000,B 0.000,C 90.000,E1 288.725} C_DIS
LIN {X -0.012,Y -406.972,Z 1495.599,A 0.000,B 0.000,C 90.000,E1 287.873} C_DIS
LIN {X -0.013,Y -413.496,Z 1495.595,A 0.000,B 0.000,C 90.000,E1 287.040} C_DIS
LIN {X 0.057,Y -419.334,Z 1495.590,A 0.000,B 0.000,C 90.000,E1 286.205} C_DIS
LIN {X 0.178,Y -424.496,Z 1495.586,A 0.000,B 0.000,C 90.000,E1 285.371} C_DIS
LIN {X -0.062,Y -428.940,Z 1495.581,A 0.000,B 0.000,C 90.000,E1 284.592} C_DIS
LIN {X 0.039,Y -432.610,Z 1495.577,A 0.000,B 0.000,C 90.000,E1 283.772} C_DIS
LIN {X -0.009,Y -434.657,Z 1495.574,A 0.000,B 0.000,C 90.000,E1 283.244} C_DIS
LIN {X -0.045,Y -436.348,Z 1495.571,A 0.000,B 0.000,C 90.000,E1 282.715} C_DIS
LIN {X 0.018,Y -437.682,Z 1495.568,A 0.000,B 0.000,C 90.000,E1 282.175} C_DIS
LIN {X -0.094,Y -438.507,Z 1495.565,A 0.000,B 0.000,C 90.000,E1 281.658} C_DIS
LIN {X -0.107,Y -438.853,Z 1495.562,A 0.000,B 0.000,C 90.000,E1 281.130} C_DIS
LIN {X -0.118,Y -438.666,Z 1495.559,A 0.000,B 0.000,C 90.000,E1 280.602} C_DIS
LIN {X -0.128,Y -437.911,Z 1495.556,A 0.000,B 0.000,C 90.000,E1 280.074} C_DIS
LIN {X -0.215,Y -436.540,Z 1495.553,A 0.000,B 0.000,C 90.000,E1 279.557} C_DIS
LIN {X 0.197,Y -434.525,Z 1495.550,A 0.000,B 0.000,C 90.000,E1 278.973} C_DIS
LIN {X 0.101,Y -431.731,Z 1495.547,A 0.000,B 0.000,C 90.000,E1 278.454} C_DIS
LIN {X -0.010,Y -428.080,Z 1495.544,A 0.000,B 0.000,C 90.000,E1 277.936} C_DIS
LIN {X -0.081,Y -423.405,Z 1495.541,A 0.000,B 0.000,C 90.000,E1 277.409} C_DIS
LIN {X 0.027,Y -420.683,Z 1495.540,A 0.000,B 0.000,C 90.000,E1 277.125} C_DIS
LIN {X 0.113,Y -414.790,Z 1495.537,A 0.000,B 0.000,C 90.000,E1 276.606} C_DIS
LIN {X -0.204,Y -408.625,Z 1495.534,A 0.000,B 0.000,C 90.000,E1 276.201} C_DIS
LIN {X -0.175,Y -402.319,Z 1495.532,A 0.000,B 0.000,C 90.000,E1 275.796} C_DIS
LIN {X 0.197,Y -395.812,Z 1495.530,A 0.000,B 0.000,C 90.000,E1 275.391} C_DIS
LIN {X -0.190,Y -386.120,Z 1495.528,A 0.000,B 0.000,C 90.000,E1 274.992} C_DIS
LIN {X 0.036,Y -373.602,Z 1495.525,A 0.000,B 0.000,C 90.000,E1 274.416} C_DIS
LIN {X 0.156,Y -363.916,Z 1495.522,A 0.000,B 0.000,C 90.000,E1 274.012} C_DIS
LIN {X 0.046,Y -347.897,Z 1495.519,A 0.000,B 0.000,C 90.000,E1 273.440} C_DIS
LIN {X -0.157,Y -337.698,Z 1495.517,A 0.000,B 0.000,C 90.000,E1 273.151} C_DIS
LIN {X 0.077,Y -324.187,Z 1495.515,A 0.000,B 0.000,C 90.000,E1 272.751} C_DIS
LIN {X 0.003,Y -312.970,Z 1495.514,A 0.000,B 0.000,C 90.000,E1 272.522} C_DIS
LIN {X -0.087,Y -300.933,Z 1495.513,A 0.000,B 0.000,C 90.000,E1 272.350} C_DIS
LIN {X -0.017,Y -290.127,Z 1495.512,A 0.000,B 0.000,C 90.000,E1 272.236} C_DIS
LIN {X 0.045,Y -278.877,Z 1495.512,A 0.000,B 0.000,C 90.000,E1 272.178} C_DIS
LIN {X 0.008,Y -181.233,Z 1495.512,A 0.000,B 0.000,C 90.000,E1 272.178} C_DIS
LIN {X -0.055,Y -181.578,Z 1495.501,A 0.000,B 0.000,C 90.000,E1 270.172} C_DIS
LIN {X -0.065,Y -180.882,Z 1495.473,A 0.000,B 0.000,C 90.000,E1 265.122} C_DIS
LIN {X -0.006,Y -179.002,Z 1495.445,A 0.000,B 0.000,C 90.000,E1 260.038} C_DIS
LIN {X 0.088,Y -178.599,Z 1495.440,A 0.000,B 0.000,C 90.000,E1 259.162} C_DIS
LIN {X -0.019,Y -175.652,Z 1495.412,A 0.000,B 0.000,C 90.000,E1 254.102} C_DIS
LIN {X -0.013,Y -172.370,Z 1495.388,A 0.000,B 0.000,C 90.000,E1 249.826} C_DIS
LIN {X 0.001,Y -171.163,Z 1495.378,A 0.000,B 0.000,C 90.000,E1 248.103} C_DIS
LIN {X 0.046,Y -167.461,Z 1495.354,A 0.000,B 0.000,C 90.000,E1 243.768} C_DIS
LIN {X -0.021,Y -166.857,Z 1495.349,A 0.000,B 0.000,C 90.000,E1 242.922} C_DIS
LIN {X 0.043,Y -162.843,Z 1495.325,A 0.000,B 0.000,C 90.000,E1 238.535} C_DIS
LIN {X 0.018,Y -161.526,Z 1495.316,A 0.000,B 0.000,C 90.000,E1 236.786} C_DIS
LIN {X 0.059,Y -157.526,Z 1495.291,A 0.000,B 0.000,C 90.000,E1 232.351} C_DIS
LIN {X -0.009,Y -155.551,Z 1495.276,A 0.000,B 0.000,C 90.000,E1 229.703} C_DIS
LIN {X -0.074,Y -151.842,Z 1495.251,A 0.000,B 0.000,C 90.000,E1 225.243} C_DIS
LIN {X -0.060,Y -150.062,Z 1495.236,A 0.000,B 0.000,C 90.000,E1 222.528} C_DIS
LIN {X -0.025,Y -146.871,Z 1495.211,A 0.000,B 0.000,C 90.000,E1 217.971} C_DIS
LIN {X -0.036,Y -145.456,Z 1495.196,A 0.000,B 0.000,C 90.000,E1 215.231} C_DIS
LIN {X 0.077,Y -142.872,Z 1495.170,A 0.000,B 0.000,C 90.000,E1 210.590} C_DIS
LIN {X 0.002,Y -141.490,Z 1495.150,A 0.000,B 0.000,C 90.000,E1 206.924} C_DIS
LIN {X -0.013,Y -139.385,Z 1495.114,A 0.000,B 0.000,C 90.000,E1 200.429} C_DIS
LIN {X -0.023,Y -138.841,Z 1495.098,A 0.000,B 0.000,C 90.000,E1 197.638} C_DIS
LIN {X 0.037,Y -138.354,Z 1495.056,A 0.000,B 0.000,C 90.000,E1 190.141} C_DIS
LIN {X 0.032,Y -139.520,Z 1495.005,A 0.000,B 0.000,C 90.000,E1 180.802} C_DIS
LIN {X -0.027,Y -141.182,Z 1494.974,A 0.000,B 0.000,C 90.000,E1 175.241} C_DIS
LIN {X -0.056,Y -142.561,Z 1494.958,A 0.000,B 0.000,C 90.000,E1 172.470} C_DIS
LIN {X 0.010,Y -144.843,Z 1494.932,A 0.000,B 0.000,C 90.000,E1 167.825} C_DIS
LIN {X -0.004,Y -147.467,Z 1494.912,A 0.000,B 0.000,C 90.000,E1 164.157} C_DIS
LIN {X 0.023,Y -150.051,Z 1494.892,A 0.000,B 0.000,C 90.000,E1 160.496} C_DIS
LIN {X 0.028,Y -153.395,Z 1494.872,A 0.000,B 0.000,C 90.000,E1 156.869} C_DIS
LIN {X 0.074,Y -155.925,Z 1494.857,A 0.000,B 0.000,C 90.000,E1 154.152} C_DIS
LIN {X 0.049,Y -159.792,Z 1494.837,A 0.000,B 0.000,C 90.000,E1 150.589} C_DIS
LIN {X 0.034,Y -162.032,Z 1494.827,A 0.000,B 0.000,C 90.000,E1 148.820} C_DIS
LIN {X 0.009,Y -166.226,Z 1494.807,A 0.000,B 0.000,C 90.000,E1 145.308} C_DIS
LIN {X 0.010,Y -171.243,Z 1494.788,A 0.000,B 0.000,C 90.000,E1 141.823} C_DIS
LIN {X -0.067,Y -176.132,Z 1494.769,A 0.000,B 0.000,C 90.000,E1 138.405} C_DIS
LIN {X 0.049,Y -180.397,Z 1494.755,A 0.000,B 0.000,C 90.000,E1 135.810} C_DIS
LIN {X 0.026,Y -185.805,Z 1494.736,A 0.000,B 0.000,C 90.000,E1 132.447} C_DIS
LIN {X 0.081,Y -190.423,Z 1494.722,A 0.000,B 0.000,C 90.000,E1 129.930} C_DIS
LIN {X -0.028,Y -197.748,Z 1494.699,A 0.000,B 0.000,C 90.000,E1 125.851} C_DIS
LIN {X -0.094,Y -201.418,Z 1494.689,A 0.000,B 0.000,C 90.000,E1 123.992} C_DIS
LIN {X -0.044,Y -201.666,Z 1494.688,A 0.000,B 0.000,C 90.000,E1 123.833} C_DIS
LIN {X -0.102,Y -314.647,Z 1494.688,A 0.000,B 0.000,C 90.000,E1 123.833} C_DIS
LIN {X 0.093,Y -315.875,Z 1494.688,A 0.000,B 0.000,C 90.000,E1 123.785} C_DIS
LIN {X 0.148,Y -320.950,Z 1494.687,A 0.000,B 0.000,C 90.000,E1 123.579} C_DIS
LIN {X -0.067,Y -323.502,Z 1494.686,A 0.000,B 0.000,C 90.000,E1 123.420} C_DIS
LIN {X -0.024,Y -327.313,Z 1494.683,A 0.000,B 0.000,C 90.000,E1 122.959} C_DIS
LIN {X 0.083,Y -329.151,Z 1494.681,A 0.000,B 0.000,C 90.000,E1 122.625} C_DIS
LIN {X -0.088,Y -330.582,Z 1494.680,A 0.000,B 0.000,C 90.000,E1 122.339} C_DIS
LIN {X 0.014,Y -342.791,Z 1494.662,A 0.000,B 0.000,C 90.000,E1 119.205} C_DIS
LIN {X -0.182,Y -355.212,Z 1494.647,A 0.000,B 0.000,C 90.000,E1 116.488} C_DIS
LIN {X -0.022,Y -369.127,Z 1494.632,A 0.000,B 0.000,C 90.000,E1 113.770} C_DIS
LIN {X 0.124,Y -382.843,Z 1494.619,A 0.000,B 0.000,C 90.000,E1 111.408} C_DIS
LIN {X -0.031,Y -397.927,Z 1494.606,A 0.000,B 0.000,C 90.000,E1 109.141} C_DIS
LIN {X -0.085,Y -414.483,Z 1494.594,A 0.000,B 0.000,C 90.000,E1 106.913} C_DIS
LIN {X 0.037,Y -432.628,Z 1494.582,A 0.000,B 0.000,C 90.000,E1 104.717} C_DIS
LIN {X -0.183,Y -452.270,Z 1494.570,A 0.000,B 0.000,C 90.000,E1 102.647} C_DIS
LIN {X 0.251,Y -472.564,Z 1494.559,A 0.000,B 0.000,C 90.000,E1 100.658} C_DIS
LIN {X -0.223,Y -490.554,Z 1494.551,A 0.000,B 0.000,C 90.000,E1 99.151} C_DIS
LIN {X -0.054,Y -492.409,Z 1494.549,A 0.000,B 0.000,C 90.000,E1 98.916} C_DIS
LIN {X -0.149,Y -494.015,Z 1494.548,A 0.000,B 0.000,C 90.000,E1 98.681} C_DIS
LIN {X 0.171,Y -495.212,Z 1494.547,A 0.000,B 0.000,C 90.000,E1 98.398} C_DIS
LIN {X -0.071,Y -496.654,Z 1494.544,A 0.000,B 0.000,C 90.000,E1 97.936} C_DIS
LIN {X 0.250,Y -497.035,Z 1494.541,A 0.000,B 0.000,C 90.000,E1 97.409} C_DIS
LIN {X 0.020,Y -496.423,Z 1494.539,A 0.000,B 0.000,C 90.000,E1 96.947} C_DIS
LIN {X -0.208,Y -494.719,Z 1494.536,A 0.000,B 0.000,C 90.000,E1 96.486} C_DIS
LIN {X 0.140,Y -493.360,Z 1494.535,A 0.000,B 0.000,C 90.000,E1 96.201} C_DIS
LIN {X -0.021,Y -484.999,Z 1494.528,A 0.000,B 0.000,C 90.000,E1 94.992} C_DIS
LIN {X 0.144,Y -472.895,Z 1494.517,A 0.000,B 0.000,C 90.000,E1 92.980} C_DIS
LIN {X 0.133,Y -464.814,Z 1494.510,A 0.000,B 0.000,C 90.000,E1 91.718} C_DIS
LIN {X -0.224,Y -454.638,Z 1494.501,A 0.000,B 0.000,C 90.000,E1 90.229} C_DIS
LIN {X 0.155,Y -444.138,Z 1494.492,A 0.000,B 0.000,C 90.000,E1 88.625} C_DIS
LIN {X -0.088,Y -433.517,Z 1494.484,A 0.000,B 0.000,C 90.000,E1 87.078} C_DIS
LIN {X 0.206,Y -419.322,Z 1494.472,A 0.000,B 0.000,C 90.000,E1 84.894} C_DIS
LIN {X 0.094,Y -406.862,Z 1494.461,A 0.000,B 0.000,C 90.000,E1 82.996} C_DIS
LIN {X -0.097,Y -392.523,Z 1494.449,A 0.000,B 0.000,C 90.000,E1 80.792} C_DIS
LIN {X -0.108,Y -373.507,Z 1494.431,A 0.000,B 0.000,C 90.000,E1 77.645} C_DIS
LIN {X 0.012,Y -362.138,Z 1494.420,A 0.000,B 0.000,C 90.000,E1 75.574} C_DIS
LIN {X -0.113,Y -350.884,Z 1494.408,A 0.000,B 0.000,C 90.000,E1 73.504} C_DIS
LIN {X 0.048,Y -339.595,Z 1494.396,A 0.000,B 0.000,C 90.000,E1 71.348} C_DIS
LIN {X 0.105,Y -325.409,Z 1494.381,A 0.000,B 0.000,C 90.000,E1 68.539} C_DIS
LIN {X -0.017,Y -309.097,Z 1494.361,A 0.000,B 0.000,C 90.000,E1 65.049} C_DIS
LIN {X -0.028,Y -296.642,Z 1494.345,A 0.000,B 0.000,C 90.000,E1 62.103} C_DIS
LIN {X 0.039,Y -284.799,Z 1494.328,A 0.000,B 0.000,C 90.000,E1 59.076} C_DIS
LIN {X 0.034,Y -274.711,Z 1494.313,A 0.000,B 0.000,C 90.000,E1 56.342} C_DIS
LIN {X -0.001,Y -263.784,Z 1494.296,A 0.000,B 0.000,C 90.000,E1 53.210} C_DIS
LIN {X 0.102,Y -252.276,Z 1494.276,A 0.000,B 0.000,C 90.000,E1 49.622} C_DIS
LIN {X -0.011,Y -242.658,Z 1494.258,A 0.000,B 0.000,C 90.000,E1 46.377} C_DIS
LIN {X -0.012,Y -234.714,Z 1494.241,A 0.000,B 0.000,C 90.000,E1 43.419} C_DIS
LIN {X 0.028,Y -225.821,Z 1494.220,A 0.000,B 0.000,C 90.000,E1 39.644} C_DIS
LIN {X 0.025,Y -219.401,Z 1494.203,A 0.000,B 0.000,C 90.000,E1 36.583} C_DIS
LIN {X 0.006,Y -212.246,Z 1494.182,A 0.000,B 0.000,C 90.000,E1 32.704} C_DIS
LIN {X 0.074,Y -205.977,Z 1494.160,A 0.000,B 0.000,C 90.000,E1 28.743} C_DIS
LIN {X -0.008,Y -200.624,Z 1494.138,A 0.000,B 0.000,C 90.000,E1 24.771} C_DIS
LIN {X -0.030,Y -196.062,Z 1494.115,A 0.000,B 0.000,C 90.000,E1 20.737} C_DIS
LIN {X 0.087,Y -192.210,Z 1494.093,A 0.000,B 0.000,C 90.000,E1 16.622} C_DIS
LIN {X -0.021,Y -188.653,Z 1494.065,A 0.000,B 0.000,C 90.000,E1 11.715} C_DIS
LIN {X -0.034,Y -185.904,Z 1494.033,A 0.000,B 0.000,C 90.000,E1 5.910} C_DIS
LIN {X -0.063,Y -184.408,Z 1493.988,A 0.000,B 0.000,C 90.000,E1 357.879} C_DIS
LIN {X -0.002,Y -185.024,Z 1493.956,A 0.000,B 0.000,C 90.000,E1 352.008} C_DIS
LIN {X -0.008,Y -187.375,Z 1493.919,A 0.000,B 0.000,C 90.000,E1 345.338} C_DIS
LIN {X -0.029,Y -190.644,Z 1493.891,A 0.000,B 0.000,C 90.000,E1 340.369} C_DIS
LIN {X 0.051,Y -194.239,Z 1493.868,A 0.000,B 0.000,C 90.000,E1 336.230} C_DIS
LIN {X 0.033,Y -198.716,Z 1493.845,A 0.000,B 0.000,C 90.000,E1 332.153} C_DIS
LIN {X 0.005,Y -204.230,Z 1493.823,A 0.000,B 0.000,C 90.000,E1 328.122} C_DIS
LIN {X 0.119,Y -209.494,Z 1493.805,A 0.000,B 0.000,C 90.000,E1 324.895} C_DIS
LIN {X -0.036,Y -215.539,Z 1493.788,A 0.000,B 0.000,C 90.000,E1 321.778} C_DIS
LIN {X 0.017,Y -222.439,Z 1493.770,A 0.000,B 0.000,C 90.000,E1 318.647} C_DIS
LIN {X 0.057,Y -230.359,Z 1493.753,A 0.000,B 0.000,C 90.000,E1 315.567} C_DIS
LIN {X 0.002,Y -239.212,Z 1493.736,A 0.000,B 0.000,C 90.000,E1 312.567} C_DIS
LIN {X -0.155,Y -249.106,Z 1493.720,A 0.000,B 0.000,C 90.000,E1 309.644} C_DIS
LIN {X -0.089,Y -256.081,Z 1493.710,A 0.000,B 0.000,C 90.000,E1 307.810} C_DIS
LIN {X -0.070,Y -263.893,Z 1493.700,A 0.000,B 0.000,C 90.000,E1 306.011} C_DIS
LIN {X -0.152,Y -270.719,Z 1493.692,A 0.000,B 0.000,C 90.000,E1 304.612} C_DIS
LIN {X 0.025,Y -280.190,Z 1493.682,A 0.000,B 0.000,C 90.000,E1 302.832} C_DIS
LIN {X -0.056,Y -292.776,Z 1493.671,A 0.000,B 0.000,C 90.000,E1 300.797} C_DIS
LIN {X -0.084,Y -302.001,Z 1493.664,A 0.000,B 0.000,C 90.000,E1 299.461} C_DIS
LIN {X 0.128,Y -312.245,Z 1493.656,A 0.000,B 0.000,C 90.000,E1 298.103} C_DIS
LIN {X -0.102,Y -334.168,Z 1493.642,A 0.000,B 0.000,C 90.000,E1 295.668} C_DIS
LIN {X -0.130,Y -353.387,Z 1493.631,A 0.000,B 0.000,C 90.000,E1 293.695} C_DIS
LIN {X -0.169,Y -366.801,Z 1493.624,A 0.000,B 0.000,C 90.000,E1 292.333} C_DIS
LIN {X -0.012,Y -377.214,Z 1493.618,A 0.000,B 0.000,C 90.000,E1 291.227} C_DIS
LIN {X 0.161,Y -390.116,Z 1493.610,A 0.000,B 0.000,C 90.000,E1 289.812} C_DIS
LIN {X -0.069,Y -400.147,Z 1493.604,A 0.000,B 0.000,C 90.000,E1 288.725} C_DIS
LIN {X 0.000,Y -407.197,Z 1493.599,A 0.000,B 0.000,C 90.000,E1 287.873} C_DIS
LIN {X 0.002,Y -413.708,Z 1493.595,A 0.000,B 0.000,C 90.000,E1 287.040} C_DIS
LIN {X 0.074,Y -419.599,Z 1493.590,A 0.000,B 0.000,C 90.000,E1 286.205} C_DIS
LIN {X -0.212,Y -424.804,Z 1493.586,A 0.000,B 0.000,C 90.000,E1 285.426} C_DIS
LIN {X -0.040,Y -429.256,Z 1493.581,A 0.000,B 0.000,C 90.000,E1 284.592} C_DIS
LIN {X 0.064,Y -432.946,Z 1493.577,A 0.000,B 0.000,C 90.000,E1 283.772} C_DIS
LIN {X 0.017,Y -435.017,Z 1493.574,A 0.000,B 0.000,C 90.000,E1 283.244} C_DIS
LIN {X -0.016,Y -436.765,Z 1493.571,A 0.000,B 0.000,C 90.000,E1 282.715} C_DIS
LIN {X -0.043,Y -438.095,Z 1493.568,A 0.000,B 0.000,C 90.000,E1 282.187} C_DIS
LIN {X -0.060,Y -438.936,Z 1493.565,A 0.000,B 0.000,C 90.000,E1 281.658} C_DIS
LIN {X -0.071,Y -439.312,Z 1493.562,A 0.000,B 0.000,C 90.000,E1 281.130} C_DIS
LIN {X -0.078,Y -439.158,Z 1493.559,A 0.000,B 0.000,C 90.000,E1 280.602} C_DIS
LIN {X -0.086,Y -438.438,Z 1493.556,A 0.000,B 0.000,C 90.000,E1 280.074} C_DIS
LIN {X -0.171,Y -437.117,Z 1493.553,A 0.000,B 0.000,C 90.000,E1 279.557} C_DIS
LIN {X -0.186,Y -435.122,Z 1493.550,A 0.000,B 0.000,C 90.000,E1 279.029} C_DIS
LIN {X 0.151,Y -432.392,Z 1493.547,A 0.000,B 0.000,C 90.000,E1 278.454} C_DIS
LIN {X 0.043,Y -428.775,Z 1493.544,A 0.000,B 0.000,C 90.000,E1 277.936} C_DIS
LIN {X -0.025,Y -424.139,Z 1493.541,A 0.000,B 0.000,C 90.000,E1 277.409} C_DIS
LIN {X -0.170,Y -418.462,Z 1493.538,A 0.000,B 0.000,C 90.000,E1 276.891} C_DIS
LIN {X 0.104,Y -412.371,Z 1493.536,A 0.000,B 0.000,C 90.000,E1 276.372} C_DIS
LIN {X -0.013,Y -406.193,Z 1493.533,A 0.000,B 0.000,C 90.000,E1 275.967} C_DIS
LIN {X 0.115,Y -399.650,Z 1493.531,A 0.000,B 0.000,C 90.000,E1 275.568} C_DIS
LIN {X -0.001,Y -389.931,Z 1493.528,A 0.000,B 0.000,C 90.000,E1 275.106} C_DIS
LIN {X 0.121,Y -377.259,Z 1493.525,A 0.000,B 0.000,C 90.000,E1 274.531} C_DIS
LIN {X 0.127,Y -364.484,Z 1493.522,A 0.000,B 0.000,C 90.000,E1 274.012} C_DIS
LIN {X 0.036,Y -348.504,Z 1493.519,A 0.000,B 0.000,C 90.000,E1 273.440} C_DIS
LIN {X -0.144,Y -338.395,Z 1493.517,A 0.000,B 0.000,C 90.000,E1 273.151} C_DIS
LIN {X 0.063,Y -324.834,Z 1493.515,A 0.000,B 0.000,C 90.000,E1 272.751} C_DIS
LIN {X 0.024,Y -313.838,Z 1493.514,A 0.000,B 0.000,C 90.000,E1 272.522} C_DIS
LIN {X -0.068,Y -301.697,Z 1493.513,A 0.000,B 0.000,C 90.000,E1 272.350} C_DIS
LIN {X 0.002,Y -291.210,Z 1493.512,A 0.000,B 0.000,C 90.000,E1 272.236} C_DIS
LIN {X 0.059,Y -280.523,Z 1493.512,A 0.000,B 0.000,C 90.000,E1 272.178} C_DIS
LIN {X 0.018,Y -181.233,Z 1493.512,A 0.000,B 0.000,C 90.000,E1 272.178} C_DIS
LIN {X -0.046,Y -181.578,Z 1493.501,A 0.000,B 0.000,C 90.000,E1 270.172} C_DIS
LIN {X -0.056,Y -180.882,Z 1493.473,A 0.000,B 0.000,C 90.000,E1 265.122} C_DIS
LIN {X 0.003,Y -179.002,Z 1493.445,A 0.000,B 0.000,C 90.000,E1 260.038} C_DIS
LIN {X -0.078,Y -178.601,Z 1493.440,A 0.000,B 0.000,C 90.000,E1 259.218} C_DIS
LIN {X -0.010,Y -175.653,Z 1493.412,A 0.000,B 0.000,C 90.000,E1 254.102} C_DIS
LIN {X -0.004,Y -172.372,Z 1493.388,A 0.000,B 0.000,C 90.000,E1 249.826} C_DIS
LIN {X 0.010,Y -171.166,Z 1493.378,A 0.000,B 0.000,C 90.000,E1 248.103} C_DIS
LIN {X 0.053,Y -167.463,Z 1493.354,A 0.000,B 0.000,C 90.000,E1 243.768} C_DIS
LIN {X -0.013,Y -166.860,Z 1493.349,A 0.000,B 0.000,C 90.000,E1 242.922} C_DIS
LIN {X 0.042,Y -162.164,Z 1493.320,A 0.000,B 0.000,C 90.000,E1 237.661} C_DIS
LIN {X -0.037,Y -160.724,Z 1493.311,A 0.000,B 0.000,C 90.000,E1 235.928} C_DIS
LIN {X -0.058,Y -157.529,Z 1493.291,A 0.000,B 0.000,C 90.000,E1 232.396} C_DIS
LIN {X -0.001,Y -155.554,Z 1493.276,A 0.000,B 0.000,C 90.000,E1 229.703} C_DIS
LIN {X -0.067,Y -151.844,Z 1493.251,A 0.000,B 0.000,C 90.000,E1 225.243} C_DIS
LIN {X -0.052,Y -150.063,Z 1493.236,A 0.000,B 0.000,C 90.000,E1 222.528} C_DIS
LIN {X -0.018,Y -146.873,Z 1493.211,A 0.000,B 0.000,C 90.000,E1 217.971} C_DIS
LIN {X -0.028,Y -145.458,Z 1493.196,A 0.000,B 0.000,C 90.000,E1 215.231} C_DIS
LIN {X 0.084,Y -142.874,Z 1493.170,A 0.000,B 0.000,C 90.000,E1 210.590} C_DIS
LIN {X 0.011,Y -141.491,Z 1493.150,A 0.000,B 0.000,C 90.000,E1 206.924} C_DIS
LIN {X -0.004,Y -139.386,Z 1493.114,A 0.000,B 0.000,C 90.000,E1 200.429} C_DIS
LIN {X -0.016,Y -138.841,Z 1493.098,A 0.000,B 0.000,C 90.000,E1 197.638} C_DIS
LIN {X 0.044,Y -138.354,Z 1493.056,A 0.000,B 0.000,C 90.000,E1 190.141} C_DIS
LIN {X 0.040,Y -139.520,Z 1493.005,A 0.000,B 0.000,C 90.000,E1 180.802} C_DIS
LIN {X -0.019,Y -141.181,Z 1492.974,A 0.000,B 0.000,C 90.000,E1 175.241} C_DIS
LIN {X -0.048,Y -142.559,Z 1492.958,A 0.000,B 0.000,C 90.000,E1 172.470} C_DIS
LIN {X 0.017,Y -144.841,Z 1492.932,A 0.000,B 0.000,C 90.000,E1 167.825} C_DIS
LIN {X 0.005,Y -147.465,Z 1492.912,A 0.000,B 0.000,C 90.000,E1 164.157} C_DIS
LIN {X 0.031,Y -150.048,Z 1492.892,A 0.000,B 0.000,C 90.000,E1 160.496} C_DIS
LIN {X 0.036,Y -153.391,Z 1492.872,A 0.000,B 0.000,C 90.000,E1 156.869} C_DIS
LIN {X 0.083,Y -155.922,Z 1492.857,A 0.000,B 0.000,C 90.000,E1 154.152} C_DIS
LIN {X 0.057,Y -159.788,Z 1492.837,A 0.000,B 0.000,C 90.000,E1 150.589} C_DIS
LIN {X -0.095,Y -162.028,Z 1492.827,A 0.000,B 0.000,C 90.000,E1 148.869} C_DIS
LIN {X 0.017,Y -166.223,Z 1492.807,A 0.000,B 0.000,C 90.000,E1 145.308} C_DIS
LIN {X 0.020,Y -171.239,Z 1492.788,A 0.000,B 0.000,C 90.000,E1 141.823} C_DIS
LIN {X -0.058,Y -176.127,Z 1492.769,A 0.000,B 0.000,C 90.000,E1 138.405} C_DIS
LIN {X 0.059,Y -180.393,Z 1492.755,A 0.000,B 0.000,C 90.000,E1 135.810} C_DIS
LIN {X 0.035,Y -185.801,Z 1492.736,A 0.000,B 0.000,C 90.000,E1 132.447} C_DIS
LIN {X 0.089,Y -190.418,Z 1492.722,A 0.000,B 0.000,C 90.000,E1 129.930} C_DIS
LIN {X -0.018,Y -197.742,Z 1492.699,A 0.000,B 0.000,C 90.000,E1 125.851} C_DIS
LIN {X -0.084,Y -201.413,Z 1492.689,A 0.000,B 0.000,C 90.000,E1 123.992} C_DIS
LIN {X 0.053,Y -201.619,Z 1492.688,A 0.000,B 0.000,C 90.000,E1 123.833} C_DIS
LIN {X 0.048,Y -315.127,Z 1492.688,A 0.000,B 0.000,C 90.000,E1 123.833} C_DIS
LIN {X 0.111,Y -317.078,Z 1492.688,A 0.000,B 0.000,C 90.000,E1 123.785} C_DIS
LIN {X -0.104,Y -321.256,Z 1492.687,A 0.000,B 0.000,C 90.000,E1 123.627} C_DIS
LIN {X -0.052,Y -323.678,Z 1492.686,A 0.000,B 0.000,C 90.000,E1 123.420} C_DIS
LIN {X -0.126,Y -327.500,Z 1492.683,A 0.000,B 0.000,C 90.000,E1 122.959} C_DIS
LIN {X -0.031,Y -329.274,Z 1492.681,A 0.000,B 0.000,C 90.000,E1 122.625} C_DIS
LIN {X -0.100,Y -331.811,Z 1492.678,A 0.000,B 0.000,C 90.000,E1 122.005} C_DIS
LIN {X -0.115,Y -342.860,Z 1492.662,A 0.000,B 0.000,C 90.000,E1 119.205} C_DIS
LIN {X 0.005,Y -355.292,Z 1492.647,A 0.000,B 0.000,C 90.000,E1 116.437} C_DIS
LIN {X -0.155,Y -369.218,Z 1492.632,A 0.000,B 0.000,C 90.000,E1 113.770} C_DIS
LIN {X -0.012,Y -382.945,Z 1492.619,A 0.000,B 0.000,C 90.000,E1 111.408} C_DIS
LIN {X 0.206,Y -398.042,Z 1492.606,A 0.000,B 0.000,C 90.000,E1 109.087} C_DIS
LIN {X 0.170,Y -414.612,Z 1492.594,A 0.000,B 0.000,C 90.000,E1 106.858} C_DIS
LIN {X -0.108,Y -432.771,Z 1492.582,A 0.000,B 0.000,C 90.000,E1 104.717} C_DIS
LIN {X 0.115,Y -452.421,Z 1492.570,A 0.000,B 0.000,C 90.000,E1 102.591} C_DIS
LIN {X 0.113,Y -472.722,Z 1492.559,A 0.000,B 0.000,C 90.000,E1 100.658} C_DIS
LIN {X 0.033,Y -488.283,Z 1492.552,A 0.000,B 0.000,C 90.000,E1 99.321} C_DIS
LIN {X 0.126,Y -490.662,Z 1492.551,A 0.000,B 0.000,C 90.000,E1 99.095} C_DIS
LIN {X -0.188,Y -492.464,Z 1492.549,A 0.000,B 0.000,C 90.000,E1 98.916} C_DIS
LIN {X 0.205,Y -494.029,Z 1492.548,A 0.000,B 0.000,C 90.000,E1 98.624} C_DIS
LIN {X 0.038,Y -495.195,Z 1492.547,A 0.000,B 0.000,C 90.000,E1 98.398} C_DIS
LIN {X -0.205,Y -496.586,Z 1492.544,A 0.000,B 0.000,C 90.000,E1 97.936} C_DIS
LIN {X 0.115,Y -496.924,Z 1492.541,A 0.000,B 0.000,C 90.000,E1 97.409} C_DIS
LIN {X -0.116,Y -496.268,Z 1492.539,A 0.000,B 0.000,C 90.000,E1 96.947} C_DIS
LIN {X 0.148,Y -494.510,Z 1492.536,A 0.000,B 0.000,C 90.000,E1 96.429} C_DIS
LIN {X 0.005,Y -493.117,Z 1492.534,A 0.000,B 0.000,C 90.000,E1 96.201} C_DIS
LIN {X -0.156,Y -484.746,Z 1492.528,A 0.000,B 0.000,C 90.000,E1 94.992} C_DIS
LIN {X 0.007,Y -472.668,Z 1492.517,A 0.000,B 0.000,C 90.000,E1 92.980} C_DIS
LIN {X -0.007,Y -464.565,Z 1492.510,A 0.000,B 0.000,C 90.000,E1 91.718} C_DIS
LIN {X 0.091,Y -454.405,Z 1492.501,A 0.000,B 0.000,C 90.000,E1 90.172} C_DIS
LIN {X 0.015,Y -443.904,Z 1492.492,A 0.000,B 0.000,C 90.000,E1 88.625} C_DIS
LIN {X 0.204,Y -433.313,Z 1492.484,A 0.000,B 0.000,C 90.000,E1 87.020} C_DIS
LIN {X 0.064,Y -419.168,Z 1492.472,A 0.000,B 0.000,C 90.000,E1 84.894} C_DIS
LIN {X -0.046,Y -406.752,Z 1492.461,A 0.000,B 0.000,C 90.000,E1 82.996} C_DIS
LIN {X 0.080,Y -394.204,Z 1492.450,A 0.000,B 0.000,C 90.000,E1 81.027} C_DIS
LIN {X 0.115,Y -375.115,Z 1492.433,A 0.000,B 0.000,C 90.000,E1 77.881} C_DIS
LIN {X -0.119,Y -362.080,Z 1492.420,A 0.000,B 0.000,C 90.000,E1 75.574} C_DIS
LIN {X 0.095,Y -350.830,Z 1492.408,A 0.000,B 0.000,C 90.000,E1 73.449} C_DIS
LIN {X 0.032,Y -339.526,Z 1492.396,A 0.000,B 0.000,C 90.000,E1 71.329} C_DIS
LIN {X 0.019,Y -326.886,Z 1492.382,A 0.000,B 0.000,C 90.000,E1 68.847} C_DIS
LIN {X -0.055,Y -310.438,Z 1492.363,A 0.000,B 0.000,C 90.000,E1 65.357} C_DIS
LIN {X -0.144,Y -296.583,Z 1492.345,A 0.000,B 0.000,C 90.000,E1 62.103} C_DIS
LIN {X -0.099,Y -283.496,Z 1492.326,A 0.000,B 0.000,C 90.000,E1 58.742} C_DIS
LIN {X -0.132,Y -273.454,Z 1492.311,A 0.000,B 0.000,C 90.000,E1 56.008} C_DIS
LIN {X -0.040,Y -262.612,Z 1492.294,A 0.000,B 0.000,C 90.000,E1 52.844} C_DIS
LIN {X 0.029,Y -251.211,Z 1492.274,A 0.000,B 0.000,C 90.000,E1 49.256} C_DIS
LIN {X -0.131,Y -240.681,Z 1492.253,A 0.000,B 0.000,C 90.000,E1 45.648} C_DIS
LIN {X 0.154,Y -232.972,Z 1492.237,A 0.000,B 0.000,C 90.000,E1 42.609} C_DIS
LIN {X -0.022,Y -224.301,Z 1492.216,A 0.000,B 0.000,C 90.000,E1 38.874} C_DIS
LIN {X -0.023,Y -218.062,Z 1492.199,A 0.000,B 0.000,C 90.000,E1 35.804} C_DIS
LIN {X 0.093,Y -211.079,Z 1492.177,A 0.000,B 0.000,C 90.000,E1 31.878} C_DIS
LIN {X -0.084,Y -205.034,Z 1492.155,A 0.000,B 0.000,C 90.000,E1 27.975} C_DIS
LIN {X -0.008,Y -199.887,Z 1492.133,A 0.000,B 0.000,C 90.000,E1 23.951} C_DIS
LIN {X 0.057,Y -195.476,Z 1492.111,A 0.000,B 0.000,C 90.000,E1 19.885} C_DIS
LIN {X -0.045,Y -191.136,Z 1492.083,A 0.000,B 0.000,C 90.000,E1 15.009} C_DIS
LIN {X 0.027,Y -187.602,Z 1492.051,A 0.000,B 0.000,C 90.000,E1 9.208} C_DIS
LIN {X -0.056,Y -185.204,Z 1492.014,A 0.000,B 0.000,C 90.000,E1 2.579} C_DIS
LIN {X -0.007,Y -184.781,Z 1491.974,A 0.000,B 0.000,C 90.000,E1 355.355} C_DIS
LIN {X -0.008,Y -185.900,Z 1491.942,A 0.000,B 0.000,C 90.000,E1 349.511} C_DIS
LIN {X -0.007,Y -188.545,Z 1491.909,A 0.000,B 0.000,C 90.000,E1 343.685} C_DIS
LIN {X 0.006,Y -192.169,Z 1491.882,A 0.000,B 0.000,C 90.000,E1 338.720} C_DIS
LIN {X 0.109,Y -196.096,Z 1491.859,A 0.000,B 0.000,C 90.000,E1 334.588} C_DIS
LIN {X 0.058,Y -200.938,Z 1491.836,A 0.000,B 0.000,C 90.000,E1 330.539} C_DIS
LIN {X -0.041,Y -206.885,Z 1491.814,A 0.000,B 0.000,C 90.000,E1 326.548} C_DIS
LIN {X 0.088,Y -212.549,Z 1491.796,A 0.000,B 0.000,C 90.000,E1 323.336} C_DIS
LIN {X -0.034,Y -218.998,Z 1491.779,A 0.000,B 0.000,C 90.000,E1 320.231} C_DIS
LIN {X -0.080,Y -226.420,Z 1491.762,A 0.000,B 0.000,C 90.000,E1 317.148} C_DIS
LIN {X 0.031,Y -235.939,Z 1491.743,A 0.000,B 0.000,C 90.000,E1 313.704} C_DIS
LIN {X -0.061,Y -246.685,Z 1491.724,A 0.000,B 0.000,C 90.000,E1 310.378} C_DIS
LIN {X -0.018,Y -254.794,Z 1491.712,A 0.000,B 0.000,C 90.000,E1 308.177} C_DIS
LIN {X -0.013,Y -262.403,Z 1491.702,A 0.000,B 0.000,C 90.000,E1 306.377} C_DIS
LIN {X -0.047,Y -270.815,Z 1491.692,A 0.000,B 0.000,C 90.000,E1 304.612} C_DIS
LIN {X -0.159,Y -282.253,Z 1491.681,A 0.000,B 0.000,C 90.000,E1 302.546} C_DIS
LIN {X 0.041,Y -294.991,Z 1491.669,A 0.000,B 0.000,C 90.000,E1 300.463} C_DIS
LIN {X -0.105,Y -304.389,Z 1491.662,A 0.000,B 0.000,C 90.000,E1 299.155} C_DIS
LIN {X 0.003,Y -314.663,Z 1491.655,A 0.000,B 0.000,C 90.000,E1 297.847} C_DIS
LIN {X 0.054,Y -339.422,Z 1491.640,A 0.000,B 0.000,C 90.000,E1 295.103} C_DIS
LIN {X -0.108,Y -355.848,Z 1491.630,A 0.000,B 0.000,C 90.000,E1 293.462} C_DIS
LIN {X -0.011,Y -369.250,Z 1491.623,A 0.000,B 0.000,C 90.000,E1 292.078} C_DIS
LIN {X 0.008,Y -379.772,Z 1491.616,A 0.000,B 0.000,C 90.000,E1 290.972} C_DIS
LIN {X -0.013,Y -392.695,Z 1491.609,A 0.000,B 0.000,C 90.000,E1 289.577} C_DIS
LIN {X -0.137,Y -402.630,Z 1491.603,A 0.000,B 0.000,C 90.000,E1 288.471} C_DIS
LIN {X -0.183,Y -409.529,Z 1491.598,A 0.000,B 0.000,C 90.000,E1 287.638} C_DIS
LIN {X -0.153,Y -415.877,Z 1491.593,A 0.000,B 0.000,C 90.000,E1 286.804} C_DIS
LIN {X -0.067,Y -421.589,Z 1491.589,A 0.000,B 0.000,C 90.000,E1 285.969} C_DIS
LIN {X 0.079,Y -426.586,Z 1491.584,A 0.000,B 0.000,C 90.000,E1 285.134} C_DIS
LIN {X -0.150,Y -430.810,Z 1491.580,A 0.000,B 0.000,C 90.000,E1 284.356} C_DIS
LIN {X -0.027,Y -434.303,Z 1491.575,A 0.000,B 0.000,C 90.000,E1 283.536} C_DIS
LIN {X 0.132,Y -437.076,Z 1491.571,A 0.000,B 0.000,C 90.000,E1 282.715} C_DIS
LIN {X 0.106,Y -438.434,Z 1491.568,A 0.000,B 0.000,C 90.000,E1 282.187} C_DIS
LIN {X 0.090,Y -439.351,Z 1491.565,A 0.000,B 0.000,C 90.000,E1 281.658} C_DIS
LIN {X 0.082,Y -439.734,Z 1491.562,A 0.000,B 0.000,C 90.000,E1 281.130} C_DIS
LIN {X 0.077,Y -439.661,Z 1491.559,A 0.000,B 0.000,C 90.000,E1 280.602} C_DIS
LIN {X 0.071,Y -438.979,Z 1491.556,A 0.000,B 0.000,C 90.000,E1 280.074} C_DIS
LIN {X -0.011,Y -437.727,Z 1491.553,A 0.000,B 0.000,C 90.000,E1 279.557} C_DIS
LIN {X -0.023,Y -435.775,Z 1491.550,A 0.000,B 0.000,C 90.000,E1 279.029} C_DIS
LIN {X -0.112,Y -433.114,Z 1491.547,A 0.000,B 0.000,C 90.000,E1 278.511} C_DIS
LIN {X -0.214,Y -429.562,Z 1491.544,A 0.000,B 0.000,C 90.000,E1 277.992} C_DIS
LIN {X -0.032,Y -427.455,Z 1491.543,A 0.000,B 0.000,C 90.000,E1 277.701} C_DIS
LIN {X -0.162,Y -422.372,Z 1491.540,A 0.000,B 0.000,C 90.000,E1 277.182} C_DIS
LIN {X -0.119,Y -416.546,Z 1491.537,A 0.000,B 0.000,C 90.000,E1 276.663} C_DIS
LIN {X -0.075,Y -410.319,Z 1491.534,A 0.000,B 0.000,C 90.000,E1 276.201} C_DIS
LIN {X -0.078,Y -403.868,Z 1491.532,A 0.000,B 0.000,C 90.000,E1 275.796} C_DIS
LIN {X 0.189,Y -397.139,Z 1491.530,A 0.000,B 0.000,C 90.000,E1 275.391} C_DIS
LIN {X 0.116,Y -387.233,Z 1491.527,A 0.000,B 0.000,C 90.000,E1 274.935} C_DIS
LIN {X -0.152,Y -371.384,Z 1491.524,A 0.000,B 0.000,C 90.000,E1 274.302} C_DIS
LIN {X 0.005,Y -361.568,Z 1491.522,A 0.000,B 0.000,C 90.000,E1 273.898} C_DIS
LIN {X -0.030,Y -348.851,Z 1491.519,A 0.000,B 0.000,C 90.000,E1 273.440} C_DIS
LIN {X 0.141,Y -338.781,Z 1491.517,A 0.000,B 0.000,C 90.000,E1 273.094} C_DIS
LIN {X 0.030,Y -325.282,Z 1491.515,A 0.000,B 0.000,C 90.000,E1 272.751} C_DIS
LIN {X 0.017,Y -314.454,Z 1491.514,A 0.000,B 0.000,C 90.000,E1 272.522} C_DIS
LIN {X -0.069,Y -302.203,Z 1491.513,A 0.000,B 0.000,C 90.000,E1 272.350} C_DIS
LIN {X -0.001,Y -291.527,Z 1491.512,A 0.000,B 0.000,C 90.000,E1 272.236} C_DIS
LIN {X 0.060,Y -279.090,Z 1491.512,A 0.000,B 0.000,C 90.000,E1 272.178} C_DIS
LIN {X 0.018,Y -181.233,Z 1491.512,A 0.000,B 0.000,C 90.000,E1 272.178} C_DIS
LIN {X -0.045,Y -181.578,Z 1491.501,A 0.000,B 0.000,C 90.000,E1 270.172} C_DIS
LIN {X -0.055,Y -180.883,Z 1491.473,A 0.000,B 0.000,C 90.000,E1 265.122} C_DIS
LIN {X 0.004,Y -179.002,Z 1491.445,A 0.000,B 0.000,C 90.000,E1 260.038} C_DIS
LIN {X -0.077,Y -178.602,Z 1491.440,A 0.000,B 0.000,C 90.000,E1 259.218} C_DIS
LIN {X -0.009,Y -175.654,Z 1491.412,A 0.000,B 0.000,C 90.000,E1 254.102} C_DIS
LIN {X -0.003,Y -172.372,Z 1491.388,A 0.000,B 0.000,C 90.000,E1 249.826} C_DIS
LIN {X 0.011,Y -171.166,Z 1491.378,A 0.000,B 0.000,C 90.000,E1 248.103} C_DIS
LIN {X 0.055,Y -167.464,Z 1491.354,A 0.000,B 0.000,C 90.000,E1 243.768} C_DIS
LIN {X -0.012,Y -166.860,Z 1491.349,A 0.000,B 0.000,C 90.000,E1 242.922} C_DIS
LIN {X 0.042,Y -162.164,Z 1491.320,A 0.000,B 0.000,C 90.000,E1 237.661} C_DIS
LIN {X -0.037,Y -160.725,Z 1491.311,A 0.000,B 0.000,C 90.000,E1 235.928} C_DIS
LIN {X -0.057,Y -157.529,Z 1491.291,A 0.000,B 0.000,C 90.000,E1 232.396} C_DIS
LIN {X 0.001,Y -155.554,Z 1491.276,A 0.000,B 0.000,C 90.000,E1 229.703} C_DIS
LIN {X -0.066,Y -151.845,Z 1491.251,A 0.000,B 0.000,C 90.000,E1 225.243} C_DIS
LIN {X -0.051,Y -150.064,Z 1491.236,A 0.000,B 0.000,C 90.000,E1 222.528} C_DIS
LIN {X -0.017,Y -146.873,Z 1491.211,A 0.000,B 0.000,C 90.000,E1 217.971} C_DIS
LIN {X -0.027,Y -145.459,Z 1491.196,A 0.000,B 0.000,C 90.000,E1 215.231} C_DIS
LIN {X 0.086,Y -142.874,Z 1491.170,A 0.000,B 0.000,C 90.000,E1 210.590} C_DIS
LIN {X 0.012,Y -141.491,Z 1491.150,A 0.000,B 0.000,C 90.000,E1 206.924} C_DIS
LIN {X -0.003,Y -139.385,Z 1491.114,A 0.000,B 0.000,C 90.000,E1 200.429} C_DIS
LIN {X -0.015,Y -138.841,Z 1491.098,A 0.000,B 0.000,C 90.000,E1 197.638} C_DIS
LIN {X 0.045,Y -138.353,Z 1491.056,A 0.000,B 0.000,C 90.000,E1 190.141} C_DIS
LIN {X 0.041,Y -139.520,Z 1491.005,A 0.000,B 0.000,C 90.000,E1 180.802} C_DIS
LIN {X -0.018,Y -141.181,Z 1490.974,A 0.000,B 0.000,C 90.000,E1 175.241} C_DIS
LIN {X -0.047,Y -142.559,Z 1490.958,A 0.000,B 0.000,C 90.000,E1 172.470} C_DIS
LIN {X 0.019,Y -144.841,Z 1490.932,A 0.000,B 0.000,C 90.000,E1 167.825} C_DIS
LIN {X 0.005,Y -147.464,Z 1490.912,A 0.000,B 0.000,C 90.000,E1 164.157} C_DIS
LIN {X 0.032,Y -150.048,Z 1490.892,A 0.000,B 0.000,C 90.000,E1 160.496} C_DIS
LIN {X 0.037,Y -153.391,Z 1490.872,A 0.000,B 0.000,C 90.000,E1 156.869} C_DIS
LIN {X -0.057,Y -155.921,Z 1490.857,A 0.000,B 0.000,C 90.000,E1 154.204} C_DIS
LIN {X 0.058,Y -159.788,Z 1490.837,A 0.000,B 0.000,C 90.000,E1 150.589} C_DIS
LIN {X -0.094,Y -162.028,Z 1490.827,A 0.000,B 0.000,C 90.000,E1 148.869} C_DIS
LIN {X 0.018,Y -166.222,Z 1490.807,A 0.000,B 0.000,C 90.000,E1 145.308} C_DIS
LIN {X 0.021,Y -171.238,Z 1490.788,A 0.000,B 0.000,C 90.000,E1 141.823} C_DIS
LIN {X -0.057,Y -176.126,Z 1490.769,A 0.000,B 0.000,C 90.000,E1 138.405} C_DIS
LIN {X 0.059,Y -180.392,Z 1490.755,A 0.000,B 0.000,C 90.000,E1 135.810} C_DIS
LIN {X 0.037,Y -185.800,Z 1490.736,A 0.000,B 0.000,C 90.000,E1 132.447} C_DIS
LIN {X 0.091,Y -190.417,Z 1490.722,A 0.000,B 0.000,C 90.000,E1 129.930} C_DIS
LIN {X -0.017,Y -197.742,Z 1490.699,A 0.000,B 0.000,C 90.000,E1 125.851} C_DIS
LIN {X -0.082,Y -201.412,Z 1490.689,A 0.000,B 0.000,C 90.000,E1 123.992} C_DIS
LIN {X -0.103,Y -201.558,Z 1490.688,A 0.000,B 0.000,C 90.000,E1 123.913} C_DIS
LIN {X 0.061,Y -314.536,Z 1490.688,A 0.000,B 0.000,C 90.000,E1 123.865} C_DIS
LIN {X -0.056,Y -316.176,Z 1490.688,A 0.000,B 0.000,C 90.000,E1 123.865} C_DIS
LIN {X 0.036,Y -321.216,Z 1490.687,A 0.000,B 0.000,C 90.000,E1 123.627} C_DIS
LIN {X -0.050,Y -323.860,Z 1490.686,A 0.000,B 0.000,C 90.000,E1 123.420} C_DIS
LIN {X -0.188,Y -327.629,Z 1490.683,A 0.000,B 0.000,C 90.000,E1 122.959} C_DIS
LIN {X -0.094,Y -329.343,Z 1490.681,A 0.000,B 0.000,C 90.000,E1 122.625} C_DIS
LIN {X -0.162,Y -331.828,Z 1490.678,A 0.000,B 0.000,C 90.000,E1 122.005} C_DIS
LIN {X 0.122,Y -342.882,Z 1490.662,A 0.000,B 0.000,C 90.000,E1 119.155} C_DIS
LIN {X 0.098,Y -355.319,Z 1490.647,A 0.000,B 0.000,C 90.000,E1 116.411} C_DIS
LIN {X -0.223,Y -369.252,Z 1490.632,A 0.000,B 0.000,C 90.000,E1 113.770} C_DIS
LIN {X -0.080,Y -382.985,Z 1490.619,A 0.000,B 0.000,C 90.000,E1 111.408} C_DIS
LIN {X 0.136,Y -398.087,Z 1490.606,A 0.000,B 0.000,C 90.000,E1 109.087} C_DIS
LIN {X 0.098,Y -414.664,Z 1490.594,A 0.000,B 0.000,C 90.000,E1 106.858} C_DIS
LIN {X -0.181,Y -432.830,Z 1490.582,A 0.000,B 0.000,C 90.000,E1 104.717} C_DIS
LIN {X 0.042,Y -452.484,Z 1490.570,A 0.000,B 0.000,C 90.000,E1 102.591} C_DIS
LIN {X 0.043,Y -472.787,Z 1490.559,A 0.000,B 0.000,C 90.000,E1 100.658} C_DIS
LIN {X -0.036,Y -488.350,Z 1490.552,A 0.000,B 0.000,C 90.000,E1 99.321} C_DIS
LIN {X 0.058,Y -490.690,Z 1490.551,A 0.000,B 0.000,C 90.000,E1 99.095} C_DIS
LIN {X 0.231,Y -492.460,Z 1490.549,A 0.000,B 0.000,C 90.000,E1 98.859} C_DIS
LIN {X 0.137,Y -493.999,Z 1490.548,A 0.000,B 0.000,C 90.000,E1 98.624} C_DIS
LIN {X -0.031,Y -495.145,Z 1490.547,A 0.000,B 0.000,C 90.000,E1 98.398} C_DIS
LIN {X -0.206,Y -496.504,Z 1490.544,A 0.000,B 0.000,C 90.000,E1 97.928} C_DIS
LIN {X 0.046,Y -496.813,Z 1490.541,A 0.000,B 0.000,C 90.000,E1 97.409} C_DIS
LIN {X -0.185,Y -496.128,Z 1490.538,A 0.000,B 0.000,C 90.000,E1 96.947} C_DIS
LIN {X 0.078,Y -494.337,Z 1490.536,A 0.000,B 0.000,C 90.000,E1 96.429} C_DIS
LIN {X -0.065,Y -492.920,Z 1490.534,A 0.000,B 0.000,C 90.000,E1 96.201} C_DIS
LIN {X -0.228,Y -484.540,Z 1490.528,A 0.000,B 0.000,C 90.000,E1 94.992} C_DIS
LIN {X -0.068,Y -472.470,Z 1490.516,A 0.000,B 0.000,C 90.000,E1 92.980} C_DIS
LIN {X -0.083,Y -464.371,Z 1490.510,A 0.000,B 0.000,C 90.000,E1 91.718} C_DIS
LIN {X 0.013,Y -454.220,Z 1490.501,A 0.000,B 0.000,C 90.000,E1 90.172} C_DIS
LIN {X 0.128,Y -441.986,Z 1490.491,A 0.000,B 0.000,C 90.000,E1 88.339} C_DIS
LIN {X 0.016,Y -429.614,Z 1490.481,A 0.000,B 0.000,C 90.000,E1 86.502} C_DIS
LIN {X 0.088,Y -417.320,Z 1490.470,A 0.000,B 0.000,C 90.000,E1 84.609} C_DIS
LIN {X -0.022,Y -404.907,Z 1490.459,A 0.000,B 0.000,C 90.000,E1 82.704} C_DIS
LIN {X 0.136,Y -390.605,Z 1490.447,A 0.000,B 0.000,C 90.000,E1 80.443} C_DIS
LIN {X 0.048,Y -373.436,Z 1490.431,A 0.000,B 0.000,C 90.000,E1 77.589} C_DIS
LIN {X 0.125,Y -360.456,Z 1490.418,A 0.000,B 0.000,C 90.000,E1 75.227} C_DIS
LIN {X 0.059,Y -349.184,Z 1490.406,A 0.000,B 0.000,C 90.000,E1 73.142} C_DIS
LIN {X -0.146,Y -337.894,Z 1490.395,A 0.000,B 0.000,C 90.000,E1 71.040} C_DIS
LIN {X -0.084,Y -325.297,Z 1490.381,A 0.000,B 0.000,C 90.000,E1 68.539} C_DIS
LIN {X -0.120,Y -310.391,Z 1490.363,A 0.000,B 0.000,C 90.000,E1 65.357} C_DIS
LIN {X 0.193,Y -296.552,Z 1490.345,A 0.000,B 0.000,C 90.000,E1 62.025} C_DIS
LIN {X -0.135,Y -284.764,Z 1490.328,A 0.000,B 0.000,C 90.000,E1 59.076} C_DIS
LIN {X 0.146,Y -275.965,Z 1490.315,A 0.000,B 0.000,C 90.000,E1 56.628} C_DIS
LIN {X 0.070,Y -266.192,Z 1490.299,A 0.000,B 0.000,C 90.000,E1 53.863} C_DIS
LIN {X 0.048,Y -255.720,Z 1490.282,A 0.000,B 0.000,C 90.000,E1 50.678} C_DIS
LIN {X 0.017,Y -244.835,Z 1490.261,A 0.000,B 0.000,C 90.000,E1 47.067} C_DIS
LIN {X 0.007,Y -234.944,Z 1490.241,A 0.000,B 0.000,C 90.000,E1 43.380} C_DIS
LIN {X -0.101,Y -226.108,Z 1490.220,A 0.000,B 0.000,C 90.000,E1 39.644} C_DIS
LIN {X -0.094,Y -219.723,Z 1490.203,A 0.000,B 0.000,C 90.000,E1 36.583} C_DIS
LIN {X 0.016,Y -212.578,Z 1490.182,A 0.000,B 0.000,C 90.000,E1 32.673} C_DIS
LIN {X -0.018,Y -206.381,Z 1490.160,A 0.000,B 0.000,C 90.000,E1 28.743} C_DIS
LIN {X -0.084,Y -201.092,Z 1490.137,A 0.000,B 0.000,C 90.000,E1 24.771} C_DIS
LIN {X -0.090,Y -196.543,Z 1490.115,A 0.000,B 0.000,C 90.000,E1 20.737} C_DIS
LIN {X -0.091,Y -192.030,Z 1490.088,A 0.000,B 0.000,C 90.000,E1 15.843} C_DIS
LIN {X -0.065,Y -188.740,Z 1490.060,A 0.000,B 0.000,C 90.000,E1 10.894} C_DIS
LIN {X 0.035,Y -186.784,Z 1490.037,A 0.000,B 0.000,C 90.000,E1 6.720} C_DIS
LIN {X 0.045,Y -184.974,Z 1489.993,A 0.000,B 0.000,C 90.000,E1 358.682} C_DIS
LIN {X -0.078,Y -185.371,Z 1489.960,A 0.000,B 0.000,C 90.000,E1 352.875} C_DIS
LIN {X 0.046,Y -187.827,Z 1489.919,A 0.000,B 0.000,C 90.000,E1 345.338} C_DIS
LIN {X 0.042,Y -191.030,Z 1489.891,A 0.000,B 0.000,C 90.000,E1 340.369} C_DIS
LIN {X -0.043,Y -194.572,Z 1489.868,A 0.000,B 0.000,C 90.000,E1 336.282} C_DIS
LIN {X 0.036,Y -199.018,Z 1489.845,A 0.000,B 0.000,C 90.000,E1 332.180} C_DIS
LIN {X 0.113,Y -204.494,Z 1489.823,A 0.000,B 0.000,C 90.000,E1 328.122} C_DIS
LIN {X -0.055,Y -209.756,Z 1489.805,A 0.000,B 0.000,C 90.000,E1 324.975} C_DIS
LIN {X -0.077,Y -215.802,Z 1489.788,A 0.000,B 0.000,C 90.000,E1 321.823} C_DIS
LIN {X -0.011,Y -222.728,Z 1489.771,A 0.000,B 0.000,C 90.000,E1 318.690} C_DIS
LIN {X -0.118,Y -230.672,Z 1489.753,A 0.000,B 0.000,C 90.000,E1 315.648} C_DIS
LIN {X -0.035,Y -240.724,Z 1489.735,A 0.000,B 0.000,C 90.000,E1 312.243} C_DIS
LIN {X 0.034,Y -250.787,Z 1489.718,A 0.000,B 0.000,C 90.000,E1 309.277} C_DIS
LIN {X 0.130,Y -257.898,Z 1489.708,A 0.000,B 0.000,C 90.000,E1 307.443} C_DIS
LIN {X 0.086,Y -267.461,Z 1489.696,A 0.000,B 0.000,C 90.000,E1 305.311} C_DIS
LIN {X 0.053,Y -274.568,Z 1489.688,A 0.000,B 0.000,C 90.000,E1 303.913} C_DIS
LIN {X -0.091,Y -284.324,Z 1489.679,A 0.000,B 0.000,C 90.000,E1 302.212} C_DIS
LIN {X 0.154,Y -297.238,Z 1489.668,A 0.000,B 0.000,C 90.000,E1 300.129} C_DIS
LIN {X 0.040,Y -306.814,Z 1489.660,A 0.000,B 0.000,C 90.000,E1 298.821} C_DIS
LIN {X 0.036,Y -320.188,Z 1489.651,A 0.000,B 0.000,C 90.000,E1 297.206} C_DIS
LIN {X -0.163,Y -344.942,Z 1489.636,A 0.000,B 0.000,C 90.000,E1 294.591} C_DIS
LIN {X -0.146,Y -358.647,Z 1489.629,A 0.000,B 0.000,C 90.000,E1 293.206} C_DIS
LIN {X 0.110,Y -372.046,Z 1489.621,A 0.000,B 0.000,C 90.000,E1 291.791} C_DIS
LIN {X -0.216,Y -382.476,Z 1489.615,A 0.000,B 0.000,C 90.000,E1 290.737} C_DIS
LIN {X 0.114,Y -392.750,Z 1489.609,A 0.000,B 0.000,C 90.000,E1 289.577} C_DIS
LIN {X -0.022,Y -402.702,Z 1489.603,A 0.000,B 0.000,C 90.000,E1 288.471} C_DIS
LIN {X -0.065,Y -409.617,Z 1489.598,A 0.000,B 0.000,C 90.000,E1 287.638} C_DIS
LIN {X -0.033,Y -416.008,Z 1489.593,A 0.000,B 0.000,C 90.000,E1 286.804} C_DIS
LIN {X 0.056,Y -421.756,Z 1489.589,A 0.000,B 0.000,C 90.000,E1 285.969} C_DIS
LIN {X -0.207,Y -426.813,Z 1489.584,A 0.000,B 0.000,C 90.000,E1 285.190} C_DIS
LIN {X -0.021,Y -431.068,Z 1489.580,A 0.000,B 0.000,C 90.000,E1 284.356} C_DIS
LIN {X 0.105,Y -434.586,Z 1489.575,A 0.000,B 0.000,C 90.000,E1 283.536} C_DIS
LIN {X -0.159,Y -437.378,Z 1489.571,A 0.000,B 0.000,C 90.000,E1 282.771} C_DIS
LIN {X -0.185,Y -438.793,Z 1489.568,A 0.000,B 0.000,C 90.000,E1 282.243} C_DIS
LIN {X -0.200,Y -439.711,Z 1489.565,A 0.000,B 0.000,C 90.000,E1 281.715} C_DIS
LIN {X -0.208,Y -440.148,Z 1489.562,A 0.000,B 0.000,C 90.000,E1 281.186} C_DIS
LIN {X 0.221,Y -440.151,Z 1489.559,A 0.000,B 0.000,C 90.000,E1 280.602} C_DIS
LIN {X 0.141,Y -439.497,Z 1489.556,A 0.000,B 0.000,C 90.000,E1 280.084} C_DIS
LIN {X 0.139,Y -438.290,Z 1489.553,A 0.000,B 0.000,C 90.000,E1 279.557} C_DIS
LIN {X 0.128,Y -436.428,Z 1489.550,A 0.000,B 0.000,C 90.000,E1 279.029} C_DIS
LIN {X 0.041,Y -433.824,Z 1489.547,A 0.000,B 0.000,C 90.000,E1 278.511} C_DIS
LIN {X -0.058,Y -430.339,Z 1489.544,A 0.000,B 0.000,C 90.000,E1 277.992} C_DIS
LIN {X -0.116,Y -425.916,Z 1489.541,A 0.000,B 0.000,C 90.000,E1 277.466} C_DIS
LIN {X 0.164,Y -420.400,Z 1489.538,A 0.000,B 0.000,C 90.000,E1 276.891} C_DIS
LIN {X -0.052,Y -414.283,Z 1489.536,A 0.000,B 0.000,C 90.000,E1 276.429} C_DIS
LIN {X 0.160,Y -408.019,Z 1489.533,A 0.000,B 0.000,C 90.000,E1 275.967} C_DIS
LIN {X -0.162,Y -401.461,Z 1489.531,A 0.000,B 0.000,C 90.000,E1 275.625} C_DIS
LIN {X -0.129,Y -394.647,Z 1489.529,A 0.000,B 0.000,C 90.000,E1 275.277} C_DIS
LIN {X 0.002,Y -384.917,Z 1489.527,A 0.000,B 0.000,C 90.000,E1 274.821} C_DIS
LIN {X -0.079,Y -372.327,Z 1489.524,A 0.000,B 0.000,C 90.000,E1 274.302} C_DIS
LIN {X 0.080,Y -359.494,Z 1489.521,A 0.000,B 0.000,C 90.000,E1 273.784} C_DIS
LIN {X 0.024,Y -349.848,Z 1489.519,A 0.000,B 0.000,C 90.000,E1 273.440} C_DIS
LIN {X 0.175,Y -339.681,Z 1489.517,A 0.000,B 0.000,C 90.000,E1 273.094} C_DIS
LIN {X 0.040,Y -326.022,Z 1489.515,A 0.000,B 0.000,C 90.000,E1 272.751} C_DIS
LIN {X 0.018,Y -315.167,Z 1489.514,A 0.000,B 0.000,C 90.000,E1 272.522} C_DIS
LIN {X -0.061,Y -302.946,Z 1489.513,A 0.000,B 0.000,C 90.000,E1 272.350} C_DIS
LIN {X 0.010,Y -292.206,Z 1489.512,A 0.000,B 0.000,C 90.000,E1 272.236} C_DIS
LIN {X 0.104,Y -283.367,Z 1489.512,A 0.000,B 0.000,C 90.000,E1 272.178} C_DIS
LIN {X 0.046,Y -181.232,Z 1489.512,A 0.000,B 0.000,C 90.000,E1 272.178} C_DIS
LIN {X -0.018,Y -181.579,Z 1489.501,A 0.000,B 0.000,C 90.000,E1 270.172} C_DIS
LIN {X -0.029,Y -180.884,Z 1489.473,A 0.000,B 0.000,C 90.000,E1 265.122} C_DIS
LIN {X 0.031,Y -179.004,Z 1489.445,A 0.000,B 0.000,C 90.000,E1 260.038} C_DIS
LIN {X -0.051,Y -178.609,Z 1489.440,A 0.000,B 0.000,C 90.000,E1 259.218} C_DIS
LIN {X 0.017,Y -175.660,Z 1489.412,A 0.000,B 0.000,C 90.000,E1 254.102} C_DIS
LIN {X 0.022,Y -172.378,Z 1489.388,A 0.000,B 0.000,C 90.000,E1 249.826} C_DIS
LIN {X 0.037,Y -171.175,Z 1489.378,A 0.000,B 0.000,C 90.000,E1 248.103} C_DIS
LIN {X 0.080,Y -167.470,Z 1489.354,A 0.000,B 0.000,C 90.000,E1 243.768} C_DIS
LIN {X 0.014,Y -166.866,Z 1489.350,A 0.000,B 0.000,C 90.000,E1 242.922} C_DIS
LIN {X 0.068,Y -162.170,Z 1489.320,A 0.000,B 0.000,C 90.000,E1 237.661} C_DIS
LIN {X -0.012,Y -160.733,Z 1489.311,A 0.000,B 0.000,C 90.000,E1 235.928} C_DIS
LIN {X -0.033,Y -157.536,Z 1489.291,A 0.000,B 0.000,C 90.000,E1 232.396} C_DIS
LIN {X 0.025,Y -155.563,Z 1489.276,A 0.000,B 0.000,C 90.000,E1 229.703} C_DIS
LIN {X -0.042,Y -151.851,Z 1489.251,A 0.000,B 0.000,C 90.000,E1 225.243} C_DIS
LIN {X -0.027,Y -150.071,Z 1489.236,A 0.000,B 0.000,C 90.000,E1 222.528} C_DIS
LIN {X 0.007,Y -146.878,Z 1489.211,A 0.000,B 0.000,C 90.000,E1 217.971} C_DIS
LIN {X -0.004,Y -145.464,Z 1489.196,A 0.000,B 0.000,C 90.000,E1 215.231} C_DIS
LIN {X -0.087,Y -142.878,Z 1489.170,A 0.000,B 0.000,C 90.000,E1 210.669} C_DIS
LIN {X 0.034,Y -141.496,Z 1489.150,A 0.000,B 0.000,C 90.000,E1 206.924} C_DIS
LIN {X 0.020,Y -139.387,Z 1489.114,A 0.000,B 0.000,C 90.000,E1 200.429} C_DIS
LIN {X 0.007,Y -138.843,Z 1489.098,A 0.000,B 0.000,C 90.000,E1 197.638} C_DIS
LIN {X -0.069,Y -138.353,Z 1489.057,A 0.000,B 0.000,C 90.000,E1 190.197} C_DIS
LIN {X 0.063,Y -139.519,Z 1489.005,A 0.000,B 0.000,C 90.000,E1 180.802} C_DIS
LIN {X 0.004,Y -141.177,Z 1488.974,A 0.000,B 0.000,C 90.000,E1 175.241} C_DIS
LIN {X -0.024,Y -142.556,Z 1488.958,A 0.000,B 0.000,C 90.000,E1 172.470} C_DIS
LIN {X 0.042,Y -144.835,Z 1488.932,A 0.000,B 0.000,C 90.000,E1 167.825} C_DIS
LIN {X 0.029,Y -147.458,Z 1488.912,A 0.000,B 0.000,C 90.000,E1 164.157} C_DIS
LIN {X 0.056,Y -150.041,Z 1488.892,A 0.000,B 0.000,C 90.000,E1 160.496} C_DIS
LIN {X -0.080,Y -153.381,Z 1488.872,A 0.000,B 0.000,C 90.000,E1 156.922} C_DIS
LIN {X -0.032,Y -155.913,Z 1488.857,A 0.000,B 0.000,C 90.000,E1 154.204} C_DIS
LIN {X 0.083,Y -159.777,Z 1488.837,A 0.000,B 0.000,C 90.000,E1 150.589} C_DIS
LIN {X -0.069,Y -162.017,Z 1488.827,A 0.000,B 0.000,C 90.000,E1 148.869} C_DIS
LIN {X 0.044,Y -166.211,Z 1488.807,A 0.000,B 0.000,C 90.000,E1 145.308} C_DIS
LIN {X 0.046,Y -171.226,Z 1488.788,A 0.000,B 0.000,C 90.000,E1 141.823} C_DIS
LIN {X -0.030,Y -176.113,Z 1488.769,A 0.000,B 0.000,C 90.000,E1 138.405} C_DIS
LIN {X 0.086,Y -180.377,Z 1488.755,A 0.000,B 0.000,C 90.000,E1 135.810} C_DIS
LIN {X 0.064,Y -185.785,Z 1488.736,A 0.000,B 0.000,C 90.000,E1 132.447} C_DIS
LIN {X -0.003,Y -190.401,Z 1488.722,A 0.000,B 0.000,C 90.000,E1 129.967} C_DIS
LIN {X 0.011,Y -197.726,Z 1488.699,A 0.000,B 0.000,C 90.000,E1 125.851} C_DIS
LIN {X -0.053,Y -201.397,Z 1488.689,A 0.000,B 0.000,C 90.000,E1 123.992} C_DIS
LIN {X -0.006,Y -201.510,Z 1488.688,A 0.000,B 0.000,C 90.000,E1 123.913} C_DIS
LIN {X -0.045,Y -314.610,Z 1488.688,A 0.000,B 0.000,C 90.000,E1 123.913} C_DIS
LIN {X -0.011,Y -316.924,Z 1488.688,A 0.000,B 0.000,C 90.000,E1 123.865} C_DIS
LIN {X 0.081,Y -321.392,Z 1488.687,A 0.000,B 0.000,C 90.000,E1 123.627} C_DIS
LIN {X -0.005,Y -323.945,Z 1488.686,A 0.000,B 0.000,C 90.000,E1 123.420} C_DIS
LIN {X 0.051,Y -327.718,Z 1488.683,A 0.000,B 0.000,C 90.000,E1 122.911} C_DIS
LIN {X -0.129,Y -329.384,Z 1488.681,A 0.000,B 0.000,C 90.000,E1 122.625} C_DIS
LIN {X 0.041,Y -334.172,Z 1488.674,A 0.000,B 0.000,C 90.000,E1 121.337} C_DIS
LIN {X -0.067,Y -345.528,Z 1488.659,A 0.000,B 0.000,C 90.000,E1 118.565} C_DIS
LIN {X -0.185,Y -358.290,Z 1488.643,A 0.000,B 0.000,C 90.000,E1 115.848} C_DIS
LIN {X 0.061,Y -372.573,Z 1488.629,A 0.000,B 0.000,C 90.000,E1 113.131} C_DIS
LIN {X 0.148,Y -386.642,Z 1488.616,A 0.000,B 0.000,C 90.000,E1 110.791} C_DIS
LIN {X -0.046,Y -402.106,Z 1488.603,A 0.000,B 0.000,C 90.000,E1 108.544} C_DIS
LIN {X 0.006,Y -419.072,Z 1488.591,A 0.000,B 0.000,C 90.000,E1 106.315} C_DIS
LIN {X 0.247,Y -437.660,Z 1488.579,A 0.000,B 0.000,C 90.000,E1 104.120} C_DIS
LIN {X 0.235,Y -457.535,Z 1488.567,A 0.000,B 0.000,C 90.000,E1 102.063} C_DIS
LIN {X 0.024,Y -477.972,Z 1488.557,A 0.000,B 0.000,C 90.000,E1 100.197} C_DIS
LIN {X -0.078,Y -488.380,Z 1488.552,A 0.000,B 0.000,C 90.000,E1 99.321} C_DIS
LIN {X 0.016,Y -490.688,Z 1488.551,A 0.000,B 0.000,C 90.000,E1 99.095} C_DIS
LIN {X 0.188,Y -492.433,Z 1488.549,A 0.000,B 0.000,C 90.000,E1 98.859} C_DIS
LIN {X 0.095,Y -493.952,Z 1488.548,A 0.000,B 0.000,C 90.000,E1 98.624} C_DIS
LIN {X -0.073,Y -495.082,Z 1488.547,A 0.000,B 0.000,C 90.000,E1 98.398} C_DIS
LIN {X 0.243,Y -496.416,Z 1488.544,A 0.000,B 0.000,C 90.000,E1 97.871} C_DIS
LIN {X 0.003,Y -496.704,Z 1488.541,A 0.000,B 0.000,C 90.000,E1 97.409} C_DIS
LIN {X -0.229,Y -495.996,Z 1488.538,A 0.000,B 0.000,C 90.000,E1 96.947} C_DIS
LIN {X 0.034,Y -494.177,Z 1488.536,A 0.000,B 0.000,C 90.000,E1 96.429} C_DIS
LIN {X -0.109,Y -492.743,Z 1488.534,A 0.000,B 0.000,C 90.000,E1 96.201} C_DIS
LIN {X 0.209,Y -484.356,Z 1488.528,A 0.000,B 0.000,C 90.000,E1 94.935} C_DIS
LIN {X -0.116,Y -472.282,Z 1488.516,A 0.000,B 0.000,C 90.000,E1 92.980} C_DIS
LIN {X -0.133,Y -464.200,Z 1488.509,A 0.000,B 0.000,C 90.000,E1 91.718} C_DIS
LIN {X -0.038,Y -454.054,Z 1488.501,A 0.000,B 0.000,C 90.000,E1 90.172} C_DIS
LIN {X 0.074,Y -441.835,Z 1488.491,A 0.000,B 0.000,C 90.000,E1 88.339} C_DIS
LIN {X -0.185,Y -431.273,Z 1488.482,A 0.000,B 0.000,C 90.000,E1 86.788} C_DIS
LIN {X 0.032,Y -417.237,Z 1488.470,A 0.000,B 0.000,C 90.000,E1 84.609} C_DIS
LIN {X -0.078,Y -404.870,Z 1488.459,A 0.000,B 0.000,C 90.000,E1 82.704} C_DIS
LIN {X 0.019,Y -392.357,Z 1488.448,A 0.000,B 0.000,C 90.000,E1 80.735} C_DIS
LIN {X -0.033,Y -376.791,Z 1488.434,A 0.000,B 0.000,C 90.000,E1 78.173} C_DIS
LIN {X 0.107,Y -362.072,Z 1488.420,A 0.000,B 0.000,C 90.000,E1 75.519} C_DIS
LIN {X 0.038,Y -352.398,Z 1488.410,A 0.000,B 0.000,C 90.000,E1 73.740} C_DIS
LIN {X -0.097,Y -341.124,Z 1488.398,A 0.000,B 0.000,C 90.000,E1 71.638} C_DIS
LIN {X 0.048,Y -328.410,Z 1488.384,A 0.000,B 0.000,C 90.000,E1 69.135} C_DIS
LIN {X -0.084,Y -311.811,Z 1488.365,A 0.000,B 0.000,C 90.000,E1 65.665} C_DIS
LIN {X 0.139,Y -297.880,Z 1488.347,A 0.000,B 0.000,C 90.000,E1 62.359} C_DIS
LIN {X -0.140,Y -287.344,Z 1488.332,A 0.000,B 0.000,C 90.000,E1 59.744} C_DIS
LIN {X 0.005,Y -277.275,Z 1488.317,A 0.000,B 0.000,C 90.000,E1 56.993} C_DIS
LIN {X 0.033,Y -266.248,Z 1488.299,A 0.000,B 0.000,C 90.000,E1 53.863} C_DIS
LIN {X -0.147,Y -254.660,Z 1488.280,A 0.000,B 0.000,C 90.000,E1 50.356} C_DIS
LIN {X -0.014,Y -244.910,Z 1488.261,A 0.000,B 0.000,C 90.000,E1 47.067} C_DIS
LIN {X 0.041,Y -236.951,Z 1488.245,A 0.000,B 0.000,C 90.000,E1 44.109} C_DIS
LIN {X -0.027,Y -227.951,Z 1488.224,A 0.000,B 0.000,C 90.000,E1 40.378} C_DIS
LIN {X 0.023,Y -221.398,Z 1488.207,A 0.000,B 0.000,C 90.000,E1 37.317} C_DIS
LIN {X 0.012,Y -214.132,Z 1488.186,A 0.000,B 0.000,C 90.000,E1 33.452} C_DIS
LIN {X -0.061,Y -208.973,Z 1488.168,A 0.000,B 0.000,C 90.000,E1 30.335} C_DIS
LIN {X -0.040,Y -203.346,Z 1488.146,A 0.000,B 0.000,C 90.000,E1 26.360} C_DIS
LIN {X -0.005,Y -198.548,Z 1488.124,A 0.000,B 0.000,C 90.000,E1 22.333} C_DIS
LIN {X -0.055,Y -194.415,Z 1488.102,A 0.000,B 0.000,C 90.000,E1 18.290} C_DIS
LIN {X 0.006,Y -190.498,Z 1488.074,A 0.000,B 0.000,C 90.000,E1 13.355} C_DIS
LIN {X -0.051,Y -187.416,Z 1488.042,A 0.000,B 0.000,C 90.000,E1 7.587} C_DIS
LIN {X 0.047,Y -185.251,Z 1487.993,A 0.000,B 0.000,C 90.000,E1 358.682} C_DIS
LIN {X -0.065,Y -185.623,Z 1487.960,A 0.000,B 0.000,C 90.000,E1 352.875} C_DIS
LIN {X 0.027,Y -188.053,Z 1487.919,A 0.000,B 0.000,C 90.000,E1 345.353} C_DIS
LIN {X 0.079,Y -191.222,Z 1487.891,A 0.000,B 0.000,C 90.000,E1 340.369} C_DIS
LIN {X -0.079,Y -194.733,Z 1487.868,A 0.000,B 0.000,C 90.000,E1 336.305} C_DIS
LIN {X -0.090,Y -199.169,Z 1487.846,A 0.000,B 0.000,C 90.000,E1 332.231} C_DIS
LIN {X -0.114,Y -204.623,Z 1487.823,A 0.000,B 0.000,C 90.000,E1 328.201} C_DIS
LIN {X 0.003,Y -209.887,Z 1487.805,A 0.000,B 0.000,C 90.000,E1 324.975} C_DIS
LIN {X -0.013,Y -215.930,Z 1487.788,A 0.000,B 0.000,C 90.000,E1 321.823} C_DIS
LIN {X 0.058,Y -222.874,Z 1487.771,A 0.000,B 0.000,C 90.000,E1 318.690} C_DIS
LIN {X -0.042,Y -230.827,Z 1487.754,A 0.000,B 0.000,C 90.000,E1 315.648} C_DIS
LIN {X 0.050,Y -240.890,Z 1487.735,A 0.000,B 0.000,C 90.000,E1 312.243} C_DIS
LIN {X 0.127,Y -250.967,Z 1487.718,A 0.000,B 0.000,C 90.000,E1 309.277} C_DIS
LIN {X -0.134,Y -258.071,Z 1487.708,A 0.000,B 0.000,C 90.000,E1 307.523} C_DIS
LIN {X -0.028,Y -267.609,Z 1487.696,A 0.000,B 0.000,C 90.000,E1 305.358} C_DIS
LIN {X 0.162,Y -274.666,Z 1487.689,A 0.000,B 0.000,C 90.000,E1 303.913} C_DIS
LIN {X -0.021,Y -286.416,Z 1487.677,A 0.000,B 0.000,C 90.000,E1 301.878} C_DIS
LIN {X -0.138,Y -299.524,Z 1487.666,A 0.000,B 0.000,C 90.000,E1 299.873} C_DIS
LIN {X -0.008,Y -309.201,Z 1487.659,A 0.000,B 0.000,C 90.000,E1 298.537} C_DIS
LIN {X -0.020,Y -322.662,Z 1487.650,A 0.000,B 0.000,C 90.000,E1 296.950} C_DIS
LIN {X 0.110,Y -347.237,Z 1487.635,A 0.000,B 0.000,C 90.000,E1 294.335} C_DIS
LIN {X 0.012,Y -358.093,Z 1487.629,A 0.000,B 0.000,C 90.000,E1 293.259} C_DIS
LIN {X -0.049,Y -371.447,Z 1487.622,A 0.000,B 0.000,C 90.000,E1 291.897} C_DIS
LIN {X -0.029,Y -381.926,Z 1487.615,A 0.000,B 0.000,C 90.000,E1 290.791} C_DIS
LIN {X -0.096,Y -392.256,Z 1487.609,A 0.000,B 0.000,C 90.000,E1 289.685} C_DIS
LIN {X -0.007,Y -402.289,Z 1487.603,A 0.000,B 0.000,C 90.000,E1 288.544} C_DIS
LIN {X 0.073,Y -409.250,Z 1487.598,A 0.000,B 0.000,C 90.000,E1 287.692} C_DIS
LIN {X 0.103,Y -415.696,Z 1487.594,A 0.000,B 0.000,C 90.000,E1 286.858} C_DIS
LIN {X 0.188,Y -421.539,Z 1487.589,A 0.000,B 0.000,C 90.000,E1 286.024} C_DIS
LIN {X -0.076,Y -426.693,Z 1487.585,A 0.000,B 0.000,C 90.000,E1 285.245} C_DIS
LIN {X 0.001,Y -431.051,Z 1487.580,A 0.000,B 0.000,C 90.000,E1 284.426} C_DIS
LIN {X -0.189,Y -434.640,Z 1487.576,A 0.000,B 0.000,C 90.000,E1 283.647} C_DIS
LIN {X -0.032,Y -437.533,Z 1487.571,A 0.000,B 0.000,C 90.000,E1 282.827} C_DIS
LIN {X -0.057,Y -438.998,Z 1487.568,A 0.000,B 0.000,C 90.000,E1 282.299} C_DIS
LIN {X -0.072,Y -439.978,Z 1487.565,A 0.000,B 0.000,C 90.000,E1 281.771} C_DIS
LIN {X -0.078,Y -440.570,Z 1487.562,A 0.000,B 0.000,C 90.000,E1 281.243} C_DIS
LIN {X -0.081,Y -440.576,Z 1487.559,A 0.000,B 0.000,C 90.000,E1 280.715} C_DIS
LIN {X -0.161,Y -440.109,Z 1487.557,A 0.000,B 0.000,C 90.000,E1 280.197} C_DIS
LIN {X -0.162,Y -439.040,Z 1487.554,A 0.000,B 0.000,C 90.000,E1 279.670} C_DIS
LIN {X -0.237,Y -437.284,Z 1487.551,A 0.000,B 0.000,C 90.000,E1 279.151} C_DIS
LIN {X 0.180,Y -434.836,Z 1487.548,A 0.000,B 0.000,C 90.000,E1 278.568} C_DIS
LIN {X 0.084,Y -431.502,Z 1487.545,A 0.000,B 0.000,C 90.000,E1 278.049} C_DIS
LIN {X -0.026,Y -427.264,Z 1487.542,A 0.000,B 0.000,C 90.000,E1 277.530} C_DIS
LIN {X -0.102,Y -421.937,Z 1487.539,A 0.000,B 0.000,C 90.000,E1 277.004} C_DIS
LIN {X 0.046,Y -415.924,Z 1487.536,A 0.000,B 0.000,C 90.000,E1 276.486} C_DIS
LIN {X 0.157,Y -409.677,Z 1487.534,A 0.000,B 0.000,C 90.000,E1 276.030} C_DIS
LIN {X -0.142,Y -403.259,Z 1487.531,A 0.000,B 0.000,C 90.000,E1 275.682} C_DIS
LIN {X -0.056,Y -396.808,Z 1487.530,A 0.000,B 0.000,C 90.000,E1 275.334} C_DIS
LIN {X 0.050,Y -387.108,Z 1487.527,A 0.000,B 0.000,C 90.000,E1 274.878} C_DIS
LIN {X -0.099,Y -371.477,Z 1487.523,A 0.000,B 0.000,C 90.000,E1 274.245} C_DIS
LIN {X 0.084,Y -358.747,Z 1487.521,A 0.000,B 0.000,C 90.000,E1 273.726} C_DIS
LIN {X 0.057,Y -349.070,Z 1487.519,A 0.000,B 0.000,C 90.000,E1 273.383} C_DIS
LIN {X -0.115,Y -338.779,Z 1487.517,A 0.000,B 0.000,C 90.000,E1 273.094} C_DIS
LIN {X -0.138,Y -325.435,Z 1487.515,A 0.000,B 0.000,C 90.000,E1 272.751} C_DIS
LIN {X -0.154,Y -314.073,Z 1487.514,A 0.000,B 0.000,C 90.000,E1 272.522} C_DIS
LIN {X 0.068,Y -300.552,Z 1487.513,A 0.000,B 0.000,C 90.000,E1 272.293} C_DIS
LIN {X -0.018,Y -291.631,Z 1487.512,A 0.000,B 0.000,C 90.000,E1 272.236} C_DIS
LIN {X 0.099,Y -280.888,Z 1487.512,A 0.000,B 0.000,C 90.000,E1 272.178} C_DIS
LIN {X 0.036,Y -181.231,Z 1487.512,A 0.000,B 0.000,C 90.000,E1 272.178} C_DIS
LIN {X -0.020,Y -181.571,Z 1487.503,A 0.000,B 0.000,C 90.000,E1 270.458} C_DIS
LIN {X 0.081,Y -180.932,Z 1487.479,A 0.000,B 0.000,C 90.000,E1 266.216} C_DIS
LIN {X -0.042,Y -180.906,Z 1487.474,A 0.000,B 0.000,C 90.000,E1 265.412} C_DIS
LIN {X 0.032,Y -180.704,Z 1487.470,A 0.000,B 0.000,C 90.000,E1 264.546} C_DIS
LIN {X -0.066,Y -178.789,Z 1487.442,A 0.000,B 0.000,C 90.000,E1 259.511} C_DIS
LIN {X 0.010,Y -175.835,Z 1487.413,A 0.000,B 0.000,C 90.000,E1 254.393} C_DIS
LIN {X 0.011,Y -172.025,Z 1487.385,A 0.000,B 0.000,C 90.000,E1 249.263} C_DIS
LIN {X -0.013,Y -171.450,Z 1487.380,A 0.000,B 0.000,C 90.000,E1 248.411} C_DIS
LIN {X 0.042,Y -167.684,Z 1487.356,A 0.000,B 0.000,C 90.000,E1 244.076} C_DIS
LIN {X -0.018,Y -166.362,Z 1487.346,A 0.000,B 0.000,C 90.000,E1 242.359} C_DIS
LIN {X -0.026,Y -163.095,Z 1487.327,A 0.000,B 0.000,C 90.000,E1 238.869} C_DIS
LIN {X 0.025,Y -161.040,Z 1487.312,A 0.000,B 0.000,C 90.000,E1 236.215} C_DIS
LIN {X 0.009,Y -157.778,Z 1487.293,A 0.000,B 0.000,C 90.000,E1 232.683} C_DIS
LIN {X 0.071,Y -155.815,Z 1487.278,A 0.000,B 0.000,C 90.000,E1 229.989} C_DIS
LIN {X -0.091,Y -152.066,Z 1487.253,A 0.000,B 0.000,C 90.000,E1 225.567} C_DIS
LIN {X -0.071,Y -150.316,Z 1487.238,A 0.000,B 0.000,C 90.000,E1 222.852} C_DIS
LIN {X -0.049,Y -147.060,Z 1487.213,A 0.000,B 0.000,C 90.000,E1 218.302} C_DIS
LIN {X 0.058,Y -145.636,Z 1487.197,A 0.000,B 0.000,C 90.000,E1 215.518} C_DIS
LIN {X 0.057,Y -143.019,Z 1487.172,A 0.000,B 0.000,C 90.000,E1 210.924} C_DIS
LIN {X -0.013,Y -141.645,Z 1487.151,A 0.000,B 0.000,C 90.000,E1 207.257} C_DIS
LIN {X 0.038,Y -139.441,Z 1487.115,A 0.000,B 0.000,C 90.000,E1 200.737} C_DIS
LIN {X -0.040,Y -139.174,Z 1487.105,A 0.000,B 0.000,C 90.000,E1 198.906} C_DIS
LIN {X -0.012,Y -138.319,Z 1487.053,A 0.000,B 0.000,C 90.000,E1 189.557} C_DIS
LIN {X -0.003,Y -139.471,Z 1487.006,A 0.000,B 0.000,C 90.000,E1 181.146} C_DIS
LIN {X -0.063,Y -141.042,Z 1486.975,A 0.000,B 0.000,C 90.000,E1 175.584} C_DIS
LIN {X 0.033,Y -142.411,Z 1486.960,A 0.000,B 0.000,C 90.000,E1 172.761} C_DIS
LIN {X -0.047,Y -144.645,Z 1486.934,A 0.000,B 0.000,C 90.000,E1 168.173} C_DIS
LIN {X 0.013,Y -147.840,Z 1486.909,A 0.000,B 0.000,C 90.000,E1 163.559} C_DIS
LIN {X -0.044,Y -150.538,Z 1486.888,A 0.000,B 0.000,C 90.000,E1 159.934} C_DIS
LIN {X -0.024,Y -154.003,Z 1486.868,A 0.000,B 0.000,C 90.000,E1 156.305} C_DIS
LIN {X 0.035,Y -157.417,Z 1486.848,A 0.000,B 0.000,C 90.000,E1 152.692} C_DIS
LIN {X 0.058,Y -161.628,Z 1486.829,A 0.000,B 0.000,C 90.000,E1 149.125} C_DIS
LIN {X 0.076,Y -165.824,Z 1486.809,A 0.000,B 0.000,C 90.000,E1 145.595} C_DIS
LIN {X 0.069,Y -170.793,Z 1486.790,A 0.000,B 0.000,C 90.000,E1 142.110} C_DIS
LIN {X -0.015,Y -175.664,Z 1486.771,A 0.000,B 0.000,C 90.000,E1 138.690} C_DIS
LIN {X -0.017,Y -181.277,Z 1486.752,A 0.000,B 0.000,C 90.000,E1 135.283} C_DIS
LIN {X -0.017,Y -186.754,Z 1486.733,A 0.000,B 0.000,C 90.000,E1 131.919} C_DIS
LIN {X 0.056,Y -191.349,Z 1486.719,A 0.000,B 0.000,C 90.000,E1 129.402} C_DIS
LIN {X -0.021,Y -197.186,Z 1486.701,A 0.000,B 0.000,C 90.000,E1 126.137} C_DIS
LIN {X 0.048,Y -201.133,Z 1486.690,A 0.000,B 0.000,C 90.000,E1 124.119} C_DIS
LIN {X 0.080,Y -201.469,Z 1486.688,A 0.000,B 0.000,C 90.000,E1 123.913} C_DIS
LIN {X 0.087,Y -314.873,Z 1486.688,A 0.000,B 0.000,C 90.000,E1 123.913} C_DIS
LIN {X -0.026,Y -316.117,Z 1486.688,A 0.000,B 0.000,C 90.000,E1 123.913} C_DIS
LIN {X -0.070,Y -320.926,Z 1486.687,A 0.000,B 0.000,C 90.000,E1 123.706} C_DIS
LIN {X -0.021,Y -324.121,Z 1486.686,A 0.000,B 0.000,C 90.000,E1 123.420} C_DIS
LIN {X 0.039,Y -327.775,Z 1486.683,A 0.000,B 0.000,C 90.000,E1 122.911} C_DIS
LIN {X -0.140,Y -329.399,Z 1486.681,A 0.000,B 0.000,C 90.000,E1 122.625} C_DIS
LIN {X -0.069,Y -344.184,Z 1486.660,A 0.000,B 0.000,C 90.000,E1 118.871} C_DIS
LIN {X 0.081,Y -356.788,Z 1486.645,A 0.000,B 0.000,C 90.000,E1 116.104} C_DIS
LIN {X -0.040,Y -370.893,Z 1486.630,A 0.000,B 0.000,C 90.000,E1 113.439} C_DIS
LIN {X -0.001,Y -384.795,Z 1486.617,A 0.000,B 0.000,C 90.000,E1 111.099} C_DIS
LIN {X -0.115,Y -400.079,Z 1486.604,A 0.000,B 0.000,C 90.000,E1 108.833} C_DIS
LIN {X -0.244,Y -416.852,Z 1486.592,A 0.000,B 0.000,C 90.000,E1 106.622} C_DIS
LIN {X 0.047,Y -435.232,Z 1486.580,A 0.000,B 0.000,C 90.000,E1 104.411} C_DIS
LIN {X -0.123,Y -454.998,Z 1486.569,A 0.000,B 0.000,C 90.000,E1 102.355} C_DIS
LIN {X -0.049,Y -475.369,Z 1486.558,A 0.000,B 0.000,C 90.000,E1 100.433} C_DIS
LIN {X -0.095,Y -488.373,Z 1486.552,A 0.000,B 0.000,C 90.000,E1 99.321} C_DIS
LIN {X -0.002,Y -490.658,Z 1486.551,A 0.000,B 0.000,C 90.000,E1 99.095} C_DIS
LIN {X 0.171,Y -492.385,Z 1486.549,A 0.000,B 0.000,C 90.000,E1 98.859} C_DIS
LIN {X 0.077,Y -493.890,Z 1486.548,A 0.000,B 0.000,C 90.000,E1 98.624} C_DIS
LIN {X -0.091,Y -495.009,Z 1486.547,A 0.000,B 0.000,C 90.000,E1 98.398} C_DIS
LIN {X 0.225,Y -496.323,Z 1486.544,A 0.000,B 0.000,C 90.000,E1 97.871} C_DIS
LIN {X -0.015,Y -496.594,Z 1486.541,A 0.000,B 0.000,C 90.000,E1 97.409} C_DIS
LIN {X 0.245,Y -495.871,Z 1486.538,A 0.000,B 0.000,C 90.000,E1 96.891} C_DIS
LIN {X 0.015,Y -494.032,Z 1486.536,A 0.000,B 0.000,C 90.000,E1 96.429} C_DIS
LIN {X -0.129,Y -492.584,Z 1486.534,A 0.000,B 0.000,C 90.000,E1 96.201} C_DIS
LIN {X 0.187,Y -484.186,Z 1486.528,A 0.000,B 0.000,C 90.000,E1 94.935} C_DIS
LIN {X -0.141,Y -472.114,Z 1486.516,A 0.000,B 0.000,C 90.000,E1 92.980} C_DIS
LIN {X -0.160,Y -464.047,Z 1486.509,A 0.000,B 0.000,C 90.000,E1 91.718} C_DIS
LIN {X -0.068,Y -453.907,Z 1486.501,A 0.000,B 0.000,C 90.000,E1 90.172} C_DIS
LIN {X 0.043,Y -441.699,Z 1486.491,A 0.000,B 0.000,C 90.000,E1 88.339} C_DIS
LIN {X -0.072,Y -429.393,Z 1486.480,A 0.000,B 0.000,C 90.000,E1 86.502} C_DIS
LIN {X 0.130,Y -415.413,Z 1486.469,A 0.000,B 0.000,C 90.000,E1 84.318} C_DIS
LIN {X -0.007,Y -403.065,Z 1486.458,A 0.000,B 0.000,C 90.000,E1 82.413} C_DIS
LIN {X 0.112,Y -388.827,Z 1486.445,A 0.000,B 0.000,C 90.000,E1 80.151} C_DIS
LIN {X -0.045,Y -375.152,Z 1486.433,A 0.000,B 0.000,C 90.000,E1 77.881} C_DIS
LIN {X 0.045,Y -360.477,Z 1486.418,A 0.000,B 0.000,C 90.000,E1 75.227} C_DIS
LIN {X -0.019,Y -349.173,Z 1486.406,A 0.000,B 0.000,C 90.000,E1 73.142} C_DIS
LIN {X 0.098,Y -337.937,Z 1486.394,A 0.000,B 0.000,C 90.000,E1 70.986} C_DIS
LIN {X -0.002,Y -326.852,Z 1486.382,A 0.000,B 0.000,C 90.000,E1 68.827} C_DIS
LIN {X -0.108,Y -311.807,Z 1486.365,A 0.000,B 0.000,C 90.000,E1 65.665} C_DIS
LIN {X 0.116,Y -297.872,Z 1486.347,A 0.000,B 0.000,C 90.000,E1 62.359} C_DIS
LIN {X -0.017,Y -287.371,Z 1486.332,A 0.000,B 0.000,C 90.000,E1 59.715} C_DIS
LIN {X -0.015,Y -277.335,Z 1486.317,A 0.000,B 0.000,C 90.000,E1 56.993} C_DIS
LIN {X 0.014,Y -266.316,Z 1486.299,A 0.000,B 0.000,C 90.000,E1 53.863} C_DIS
LIN {X 0.034,Y -254.734,Z 1486.280,A 0.000,B 0.000,C 90.000,E1 50.312} C_DIS
LIN {X -0.021,Y -244.999,Z 1486.261,A 0.000,B 0.000,C 90.000,E1 47.067} C_DIS
LIN {X 0.037,Y -237.059,Z 1486.245,A 0.000,B 0.000,C 90.000,E1 44.109} C_DIS
LIN {X -0.027,Y -228.104,Z 1486.224,A 0.000,B 0.000,C 90.000,E1 40.378} C_DIS
LIN {X 0.027,Y -221.560,Z 1486.207,A 0.000,B 0.000,C 90.000,E1 37.317} C_DIS
LIN {X 0.022,Y -214.338,Z 1486.186,A 0.000,B 0.000,C 90.000,E1 33.452} C_DIS
LIN {X -0.048,Y -209.187,Z 1486.168,A 0.000,B 0.000,C 90.000,E1 30.335} C_DIS
LIN {X -0.020,Y -203.600,Z 1486.146,A 0.000,B 0.000,C 90.000,E1 26.360} C_DIS
LIN {X 0.022,Y -198.821,Z 1486.124,A 0.000,B 0.000,C 90.000,E1 22.333} C_DIS
LIN {X -0.019,Y -194.694,Z 1486.102,A 0.000,B 0.000,C 90.000,E1 18.290} C_DIS
LIN {X 0.051,Y -190.786,Z 1486.074,A 0.000,B 0.000,C 90.000,E1 13.355} C_DIS
LIN {X 0.004,Y -187.696,Z 1486.042,A 0.000,B 0.000,C 90.000,E1 7.587} C_DIS
LIN {X 0.049,Y -185.521,Z 1485.993,A 0.000,B 0.000,C 90.000,E1 358.682} C_DIS
LIN {X -0.051,Y -185.867,Z 1485.960,A 0.000,B 0.000,C 90.000,E1 352.875} C_DIS
LIN {X 0.089,Y -187.888,Z 1485.923,A 0.000,B 0.000,C 90.000,E1 346.172} C_DIS
LIN {X 0.026,Y -190.800,Z 1485.896,A 0.000,B 0.000,C 90.000,E1 341.221} C_DIS
LIN {X -0.037,Y -194.903,Z 1485.868,A 0.000,B 0.000,C 90.000,E1 336.305} C_DIS
LIN {X -0.042,Y -199.322,Z 1485.846,A 0.000,B 0.000,C 90.000,E1 332.231} C_DIS
LIN {X -0.060,Y -204.757,Z 1485.823,A 0.000,B 0.000,C 90.000,E1 328.201} C_DIS
LIN {X 0.063,Y -210.015,Z 1485.806,A 0.000,B 0.000,C 90.000,E1 324.975} C_DIS
LIN {X 0.051,Y -216.062,Z 1485.788,A 0.000,B 0.000,C 90.000,E1 321.823} C_DIS
LIN {X -0.019,Y -223.021,Z 1485.771,A 0.000,B 0.000,C 90.000,E1 318.728} C_DIS
LIN {X 0.035,Y -230.987,Z 1485.754,A 0.000,B 0.000,C 90.000,E1 315.648} C_DIS
LIN {X -0.044,Y -241.053,Z 1485.735,A 0.000,B 0.000,C 90.000,E1 312.285} C_DIS
LIN {X -0.144,Y -249.807,Z 1485.720,A 0.000,B 0.000,C 90.000,E1 309.725} C_DIS
LIN {X -0.064,Y -256.763,Z 1485.710,A 0.000,B 0.000,C 90.000,E1 307.890} C_DIS
LIN {X 0.022,Y -266.108,Z 1485.698,A 0.000,B 0.000,C 90.000,E1 305.724} C_DIS
LIN {X -0.030,Y -272.916,Z 1485.691,A 0.000,B 0.000,C 90.000,E1 304.326} C_DIS
LIN {X 0.137,Y -284.439,Z 1485.679,A 0.000,B 0.000,C 90.000,E1 302.212} C_DIS
LIN {X -0.010,Y -297.244,Z 1485.668,A 0.000,B 0.000,C 90.000,E1 300.207} C_DIS
LIN {X 0.027,Y -306.668,Z 1485.660,A 0.000,B 0.000,C 90.000,E1 298.871} C_DIS
LIN {X -0.122,Y -316.892,Z 1485.653,A 0.000,B 0.000,C 90.000,E1 297.641} C_DIS
LIN {X 0.140,Y -338.727,Z 1485.640,A 0.000,B 0.000,C 90.000,E1 295.207} C_DIS
LIN {X -0.023,Y -355.080,Z 1485.631,A 0.000,B 0.000,C 90.000,E1 293.590} C_DIS
LIN {X 0.089,Y -368.478,Z 1485.623,A 0.000,B 0.000,C 90.000,E1 292.206} C_DIS
LIN {X -0.143,Y -378.898,Z 1485.617,A 0.000,B 0.000,C 90.000,E1 291.153} C_DIS
LIN {X 0.235,Y -389.201,Z 1485.611,A 0.000,B 0.000,C 90.000,E1 289.993} C_DIS
LIN {X 0.038,Y -399.257,Z 1485.605,A 0.000,B 0.000,C 90.000,E1 288.906} C_DIS
LIN {X 0.099,Y -406.511,Z 1485.600,A 0.000,B 0.000,C 90.000,E1 288.055} C_DIS
LIN {X 0.096,Y -413.171,Z 1485.596,A 0.000,B 0.000,C 90.000,E1 287.221} C_DIS
LIN {X 0.165,Y -419.319,Z 1485.591,A 0.000,B 0.000,C 90.000,E1 286.386} C_DIS
LIN {X -0.121,Y -424.818,Z 1485.587,A 0.000,B 0.000,C 90.000,E1 285.607} C_DIS
LIN {X 0.052,Y -429.540,Z 1485.582,A 0.000,B 0.000,C 90.000,E1 284.773} C_DIS
LIN {X 0.161,Y -433.496,Z 1485.578,A 0.000,B 0.000,C 90.000,E1 283.953} C_DIS
LIN {X 0.219,Y -435.691,Z 1485.575,A 0.000,B 0.000,C 90.000,E1 283.411} C_DIS
LIN {X 0.188,Y -437.612,Z 1485.572,A 0.000,B 0.000,C 90.000,E1 282.883} C_DIS
LIN {X 0.162,Y -439.115,Z 1485.569,A 0.000,B 0.000,C 90.000,E1 282.355} C_DIS
LIN {X 0.148,Y -440.226,Z 1485.566,A 0.000,B 0.000,C 90.000,E1 281.827} C_DIS
LIN {X 0.141,Y -440.901,Z 1485.563,A 0.000,B 0.000,C 90.000,E1 281.299} C_DIS
LIN {X 0.057,Y -441.059,Z 1485.560,A 0.000,B 0.000,C 90.000,E1 280.782} C_DIS
LIN {X 0.060,Y -440.688,Z 1485.557,A 0.000,B 0.000,C 90.000,E1 280.254} C_DIS
LIN {X 0.061,Y -439.740,Z 1485.554,A 0.000,B 0.000,C 90.000,E1 279.726} C_DIS
LIN {X -0.013,Y -438.155,Z 1485.551,A 0.000,B 0.000,C 90.000,E1 279.208} C_DIS
LIN {X -0.023,Y -435.868,Z 1485.548,A 0.000,B 0.000,C 90.000,E1 278.681} C_DIS
LIN {X -0.114,Y -432.705,Z 1485.545,A 0.000,B 0.000,C 90.000,E1 278.163} C_DIS
LIN {X 0.076,Y -430.843,Z 1485.544,A 0.000,B 0.000,C 90.000,E1 277.871} C_DIS
LIN {X -0.039,Y -426.292,Z 1485.541,A 0.000,B 0.000,C 90.000,E1 277.352} C_DIS
LIN {X -0.074,Y -420.749,Z 1485.538,A 0.000,B 0.000,C 90.000,E1 276.834} C_DIS
LIN {X 0.201,Y -414.649,Z 1485.535,A 0.000,B 0.000,C 90.000,E1 276.315} C_DIS
LIN {X 0.060,Y -408.333,Z 1485.533,A 0.000,B 0.000,C 90.000,E1 275.910} C_DIS
LIN {X -0.172,Y -401.845,Z 1485.531,A 0.000,B 0.000,C 90.000,E1 275.568} C_DIS
LIN {X 0.044,Y -391.752,Z 1485.528,A 0.000,B 0.000,C 90.000,E1 275.049} C_DIS
LIN {X -0.104,Y -379.101,Z 1485.525,A 0.000,B 0.000,C 90.000,E1 274.531} C_DIS
LIN {X -0.024,Y -366.602,Z 1485.522,A 0.000,B 0.000,C 90.000,E1 274.012} C_DIS
LIN {X -0.175,Y -353.648,Z 1485.520,A 0.000,B 0.000,C 90.000,E1 273.555} C_DIS
LIN {X -0.104,Y -343.609,Z 1485.518,A 0.000,B 0.000,C 90.000,E1 273.212} C_DIS
LIN {X -0.097,Y -333.201,Z 1485.516,A 0.000,B 0.000,C 90.000,E1 272.922} C_DIS
LIN {X 0.159,Y -323.306,Z 1485.515,A 0.000,B 0.000,C 90.000,E1 272.636} C_DIS
LIN {X -0.070,Y -312.263,Z 1485.514,A 0.000,B 0.000,C 90.000,E1 272.465} C_DIS
LIN {X -0.104,Y -303.431,Z 1485.513,A 0.000,B 0.000,C 90.000,E1 272.350} C_DIS
LIN {X -0.037,Y -291.330,Z 1485.512,A 0.000,B 0.000,C 90.000,E1 272.236} C_DIS
LIN {X 0.104,Y -281.169,Z 1485.512,A 0.000,B 0.000,C 90.000,E1 272.178} C_DIS
LIN {X 0.036,Y -181.231,Z 1485.512,A 0.000,B 0.000,C 90.000,E1 272.178} C_DIS
LIN {X 0.026,Y -181.569,Z 1485.503,A 0.000,B 0.000,C 90.000,E1 270.458} C_DIS
LIN {X 0.067,Y -181.002,Z 1485.484,A 0.000,B 0.000,C 90.000,E1 267.078} C_DIS
LIN {X 0.004,Y -180.906,Z 1485.474,A 0.000,B 0.000,C 90.000,E1 265.412} C_DIS
LIN {X 0.061,Y -180.711,Z 1485.470,A 0.000,B 0.000,C 90.000,E1 264.552} C_DIS
LIN {X -0.021,Y -178.797,Z 1485.442,A 0.000,B 0.000,C 90.000,E1 259.511} C_DIS
LIN {X 0.056,Y -175.842,Z 1485.413,A 0.000,B 0.000,C 90.000,E1 254.393} C_DIS
LIN {X 0.055,Y -172.034,Z 1485.385,A 0.000,B 0.000,C 90.000,E1 249.263} C_DIS
LIN {X 0.031,Y -171.463,Z 1485.380,A 0.000,B 0.000,C 90.000,E1 248.411} C_DIS
LIN {X 0.012,Y -167.696,Z 1485.356,A 0.000,B 0.000,C 90.000,E1 244.101} C_DIS
LIN {X 0.025,Y -166.378,Z 1485.346,A 0.000,B 0.000,C 90.000,E1 242.359} C_DIS
LIN {X 0.017,Y -163.107,Z 1485.327,A 0.000,B 0.000,C 90.000,E1 238.869} C_DIS
LIN {X 0.067,Y -161.055,Z 1485.312,A 0.000,B 0.000,C 90.000,E1 236.215} C_DIS
LIN {X 0.050,Y -157.790,Z 1485.293,A 0.000,B 0.000,C 90.000,E1 232.683} C_DIS
LIN {X -0.007,Y -155.826,Z 1485.278,A 0.000,B 0.000,C 90.000,E1 230.033} C_DIS
LIN {X -0.049,Y -152.077,Z 1485.253,A 0.000,B 0.000,C 90.000,E1 225.567} C_DIS
LIN {X -0.030,Y -150.328,Z 1485.238,A 0.000,B 0.000,C 90.000,E1 222.852} C_DIS
LIN {X -0.009,Y -147.068,Z 1485.213,A 0.000,B 0.000,C 90.000,E1 218.302} C_DIS
LIN {X -0.021,Y -145.644,Z 1485.198,A 0.000,B 0.000,C 90.000,E1 215.564} C_DIS
LIN {X 0.096,Y -143.026,Z 1485.172,A 0.000,B 0.000,C 90.000,E1 210.924} C_DIS
LIN {X 0.026,Y -141.652,Z 1485.151,A 0.000,B 0.000,C 90.000,E1 207.257} C_DIS
LIN {X -0.054,Y -139.444,Z 1485.115,A 0.000,B 0.000,C 90.000,E1 200.791} C_DIS
LIN {X -0.001,Y -139.177,Z 1485.105,A 0.000,B 0.000,C 90.000,E1 198.906} C_DIS
LIN {X 0.027,Y -138.319,Z 1485.053,A 0.000,B 0.000,C 90.000,E1 189.557} C_DIS
LIN {X 0.036,Y -139.468,Z 1485.006,A 0.000,B 0.000,C 90.000,E1 181.146} C_DIS
LIN {X -0.023,Y -141.035,Z 1484.975,A 0.000,B 0.000,C 90.000,E1 175.584} C_DIS
LIN {X 0.072,Y -142.403,Z 1484.960,A 0.000,B 0.000,C 90.000,E1 172.761} C_DIS
LIN {X -0.007,Y -144.636,Z 1484.934,A 0.000,B 0.000,C 90.000,E1 168.173} C_DIS
LIN {X 0.053,Y -147.831,Z 1484.909,A 0.000,B 0.000,C 90.000,E1 163.559} C_DIS
LIN {X -0.003,Y -150.525,Z 1484.889,A 0.000,B 0.000,C 90.000,E1 159.934} C_DIS
LIN {X 0.017,Y -153.988,Z 1484.868,A 0.000,B 0.000,C 90.000,E1 156.305} C_DIS
LIN {X -0.062,Y -157.401,Z 1484.848,A 0.000,B 0.000,C 90.000,E1 152.743} C_DIS
LIN {X 0.018,Y -161.607,Z 1484.829,A 0.000,B 0.000,C 90.000,E1 149.154} C_DIS
LIN {X -0.018,Y -165.804,Z 1484.809,A 0.000,B 0.000,C 90.000,E1 145.642} C_DIS
LIN {X 0.009,Y -170.770,Z 1484.790,A 0.000,B 0.000,C 90.000,E1 142.145} C_DIS
LIN {X 0.031,Y -175.641,Z 1484.771,A 0.000,B 0.000,C 90.000,E1 138.690} C_DIS
LIN {X -0.100,Y -181.256,Z 1484.752,A 0.000,B 0.000,C 90.000,E1 135.324} C_DIS
LIN {X 0.030,Y -186.729,Z 1484.733,A 0.000,B 0.000,C 90.000,E1 131.919} C_DIS
LIN {X -0.019,Y -191.327,Z 1484.719,A 0.000,B 0.000,C 90.000,E1 129.439} C_DIS
LIN {X 0.028,Y -197.159,Z 1484.701,A 0.000,B 0.000,C 90.000,E1 126.137} C_DIS
LIN {X -0.076,Y -201.193,Z 1484.689,A 0.000,B 0.000,C 90.000,E1 124.119} C_DIS
LIN {X -0.096,Y -201.419,Z 1484.689,A 0.000,B 0.000,C 90.000,E1 123.992} C_DIS
LIN {X -0.192,Y -314.592,Z 1484.689,A 0.000,B 0.000,C 90.000,E1 123.992} C_DIS
LIN {X 0.007,Y -320.998,Z 1484.687,A 0.000,B 0.000,C 90.000,E1 123.706} C_DIS
LIN {X -0.032,Y -323.977,Z 1484.686,A 0.000,B 0.000,C 90.000,E1 123.452} C_DIS
LIN {X -0.092,Y -327.666,Z 1484.683,A 0.000,B 0.000,C 90.000,E1 122.959} C_DIS
LIN {X 0.005,Y -329.288,Z 1484.681,A 0.000,B 0.000,C 90.000,E1 122.625} C_DIS
LIN {X 0.078,Y -344.057,Z 1484.661,A 0.000,B 0.000,C 90.000,E1 118.871} C_DIS
LIN {X -0.090,Y -356.647,Z 1484.645,A 0.000,B 0.000,C 90.000,E1 116.155} C_DIS
LIN {X -0.037,Y -370.738,Z 1484.630,A 0.000,B 0.000,C 90.000,E1 113.462} C_DIS
LIN {X 0.151,Y -384.628,Z 1484.617,A 0.000,B 0.000,C 90.000,E1 111.099} C_DIS
LIN {X -0.090,Y -399.897,Z 1484.605,A 0.000,B 0.000,C 90.000,E1 108.852} C_DIS
LIN {X -0.088,Y -416.655,Z 1484.592,A 0.000,B 0.000,C 90.000,E1 106.622} C_DIS
LIN {X 0.097,Y -435.017,Z 1484.580,A 0.000,B 0.000,C 90.000,E1 104.426} C_DIS
LIN {X 0.029,Y -454.777,Z 1484.569,A 0.000,B 0.000,C 90.000,E1 102.355} C_DIS
LIN {X 0.096,Y -475.143,Z 1484.558,A 0.000,B 0.000,C 90.000,E1 100.433} C_DIS
LIN {X 0.045,Y -488.144,Z 1484.552,A 0.000,B 0.000,C 90.000,E1 99.321} C_DIS
LIN {X 0.138,Y -490.459,Z 1484.551,A 0.000,B 0.000,C 90.000,E1 99.095} C_DIS
LIN {X -0.177,Y -492.209,Z 1484.549,A 0.000,B 0.000,C 90.000,E1 98.916} C_DIS
LIN {X 0.216,Y -493.731,Z 1484.548,A 0.000,B 0.000,C 90.000,E1 98.624} C_DIS
LIN {X 0.047,Y -494.864,Z 1484.547,A 0.000,B 0.000,C 90.000,E1 98.398} C_DIS
